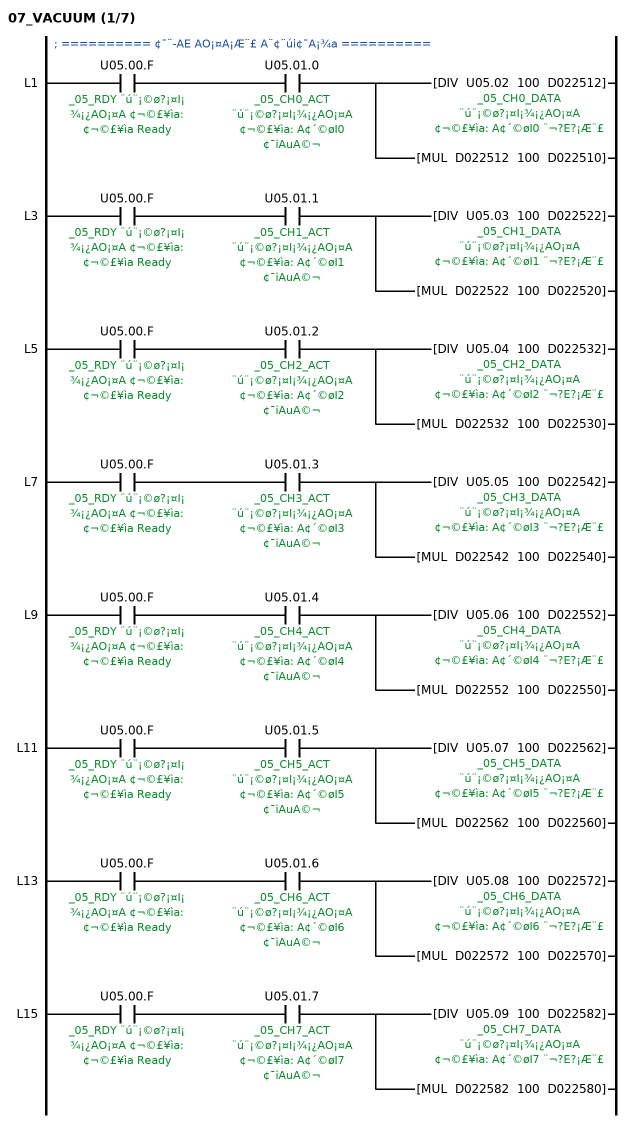
[picture p48: 07_VACUUM rungs L1-L15]
// ========== ¢¯¨­AE AO¡¤A¡Æ¨£ A¨¢¨úi¢¯A¡¾a ==========
; L1
LOAD      U05.00.F	// _05_RDY ¨ú¨¡©ø?¡¤I¡¾¡¿AO¡¤A ¢¬©£¥ìa: ¢¬©£¥ìa Ready
AND       U05.01.0	// _05_CH0_ACT ¨ú¨¡©ø?¡¤I¡¾¡¿AO¡¤A ¢¬©£¥ìa: A¢´©øI0 ¢¯iAuA©¬
DIV       U05.02 100 D022512	// _05_CH0_DATA ¨ú¨¡©ø?¡¤I¡¾¡¿AO¡¤A ¢¬©£¥ìa: A¢´©øI0 ¨¬?E?¡Æ¨£
MUL       D022512 100 D022510
; L3
LOAD      U05.00.F	// _05_RDY ¨ú¨¡©ø?¡¤I¡¾¡¿AO¡¤A ¢¬©£¥ìa: ¢¬©£¥ìa Ready
AND       U05.01.1	// _05_CH1_ACT ¨ú¨¡©ø?¡¤I¡¾¡¿AO¡¤A ¢¬©£¥ìa: A¢´©øI1 ¢¯iAuA©¬
DIV       U05.03 100 D022522	// _05_CH1_DATA ¨ú¨¡©ø?¡¤I¡¾¡¿AO¡¤A ¢¬©£¥ìa: A¢´©øI1 ¨¬?E?¡Æ¨£
MUL       D022522 100 D022520
; L5
LOAD      U05.00.F	// _05_RDY ¨ú¨¡©ø?¡¤I¡¾¡¿AO¡¤A ¢¬©£¥ìa: ¢¬©£¥ìa Ready
AND       U05.01.2	// _05_CH2_ACT ¨ú¨¡©ø?¡¤I¡¾¡¿AO¡¤A ¢¬©£¥ìa: A¢´©øI2 ¢¯iAuA©¬
DIV       U05.04 100 D022532	// _05_CH2_DATA ¨ú¨¡©ø?¡¤I¡¾¡¿AO¡¤A ¢¬©£¥ìa: A¢´©øI2 ¨¬?E?¡Æ¨£
MUL       D022532 100 D022530
; L7
LOAD      U05.00.F	// _05_RDY ¨ú¨¡©ø?¡¤I¡¾¡¿AO¡¤A ¢¬©£¥ìa: ¢¬©£¥ìa Ready
AND       U05.01.3	// _05_CH3_ACT ¨ú¨¡©ø?¡¤I¡¾¡¿AO¡¤A ¢¬©£¥ìa: A¢´©øI3 ¢¯iAuA©¬
DIV       U05.05 100 D022542	// _05_CH3_DATA ¨ú¨¡©ø?¡¤I¡¾¡¿AO¡¤A ¢¬©£¥ìa: A¢´©øI3 ¨¬?E?¡Æ¨£
MUL       D022542 100 D022540
; L9
LOAD      U05.00.F	// _05_RDY ¨ú¨¡©ø?¡¤I¡¾¡¿AO¡¤A ¢¬©£¥ìa: ¢¬©£¥ìa Ready
AND       U05.01.4	// _05_CH4_ACT ¨ú¨¡©ø?¡¤I¡¾¡¿AO¡¤A ¢¬©£¥ìa: A¢´©øI4 ¢¯iAuA©¬
DIV       U05.06 100 D022552	// _05_CH4_DATA ¨ú¨¡©ø?¡¤I¡¾¡¿AO¡¤A ¢¬©£¥ìa: A¢´©øI4 ¨¬?E?¡Æ¨£
MUL       D022552 100 D022550
; L11
LOAD      U05.00.F	// _05_RDY ¨ú¨¡©ø?¡¤I¡¾¡¿AO¡¤A ¢¬©£¥ìa: ¢¬©£¥ìa Ready
AND       U05.01.5	// _05_CH5_ACT ¨ú¨¡©ø?¡¤I¡¾¡¿AO¡¤A ¢¬©£¥ìa: A¢´©øI5 ¢¯iAuA©¬
DIV       U05.07 100 D022562	// _05_CH5_DATA ¨ú¨¡©ø?¡¤I¡¾¡¿AO¡¤A ¢¬©£¥ìa: A¢´©øI5 ¨¬?E?¡Æ¨£
MUL       D022562 100 D022560
; L13
LOAD      U05.00.F	// _05_RDY ¨ú¨¡©ø?¡¤I¡¾¡¿AO¡¤A ¢¬©£¥ìa: ¢¬©£¥ìa Ready
AND       U05.01.6	// _05_CH6_ACT ¨ú¨¡©ø?¡¤I¡¾¡¿AO¡¤A ¢¬©£¥ìa: A¢´©øI6 ¢¯iAuA©¬
DIV       U05.08 100 D022572	// _05_CH6_DATA ¨ú¨¡©ø?¡¤I¡¾¡¿AO¡¤A ¢¬©£¥ìa: A¢´©øI6 ¨¬?E?¡Æ¨£
MUL       D022572 100 D022570
; L15
LOAD      U05.00.F	// _05_RDY ¨ú¨¡©ø?¡¤I¡¾¡¿AO¡¤A ¢¬©£¥ìa: ¢¬©£¥ìa Ready
AND       U05.01.7	// _05_CH7_ACT ¨ú¨¡©ø?¡¤I¡¾¡¿AO¡¤A ¢¬©£¥ìa: A¢´©øI7 ¢¯iAuA©¬
DIV       U05.09 100 D022582	// _05_CH7_DATA ¨ú¨¡©ø?¡¤I¡¾¡¿AO¡¤A ¢¬©£¥ìa: A¢´©øI7 ¨¬?E?¡Æ¨£
MUL       D022582 100 D022580

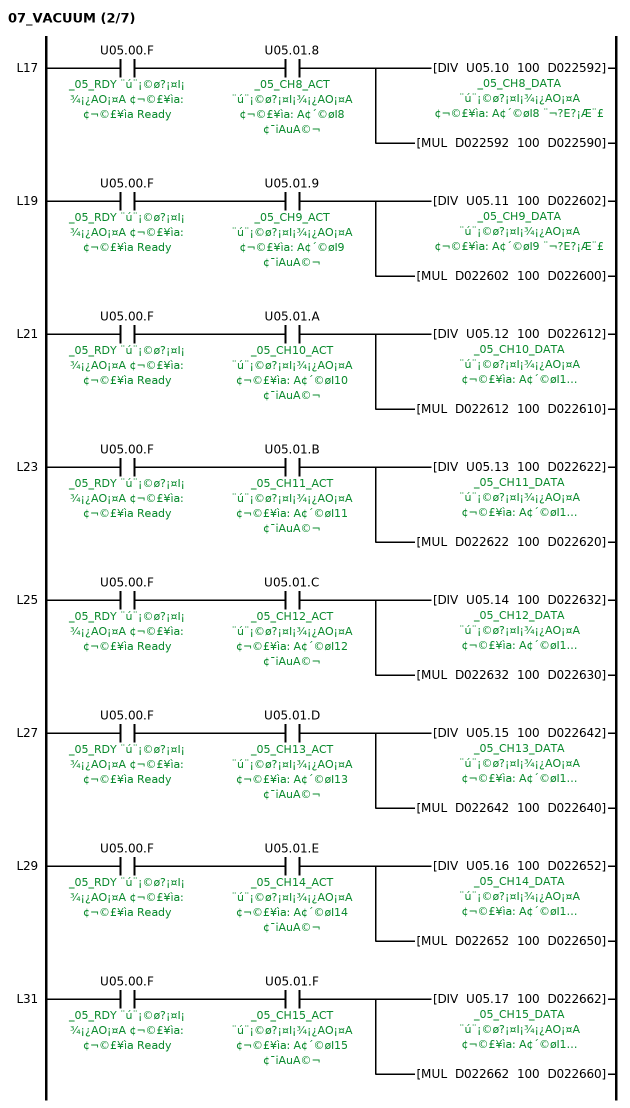
; L17
LOAD      U05.00.F	// _05_RDY ¨ú¨¡©ø?¡¤I¡¾¡¿AO¡¤A ¢¬©£¥ìa: ¢¬©£¥ìa Ready
AND       U05.01.8	// _05_CH8_ACT ¨ú¨¡©ø?¡¤I¡¾¡¿AO¡¤A ¢¬©£¥ìa: A¢´©øI8 ¢¯iAuA©¬
DIV       U05.10 100 D022592	// _05_CH8_DATA ¨ú¨¡©ø?¡¤I¡¾¡¿AO¡¤A ¢¬©£¥ìa: A¢´©øI8 ¨¬?E?¡Æ¨£
MUL       D022592 100 D022590
; L19
LOAD      U05.00.F	// _05_RDY ¨ú¨¡©ø?¡¤I¡¾¡¿AO¡¤A ¢¬©£¥ìa: ¢¬©£¥ìa Ready
AND       U05.01.9	// _05_CH9_ACT ¨ú¨¡©ø?¡¤I¡¾¡¿AO¡¤A ¢¬©£¥ìa: A¢´©øI9 ¢¯iAuA©¬
DIV       U05.11 100 D022602	// _05_CH9_DATA ¨ú¨¡©ø?¡¤I¡¾¡¿AO¡¤A ¢¬©£¥ìa: A¢´©øI9 ¨¬?E?¡Æ¨£
MUL       D022602 100 D022600
; L21
LOAD      U05.00.F	// _05_RDY ¨ú¨¡©ø?¡¤I¡¾¡¿AO¡¤A ¢¬©£¥ìa: ¢¬©£¥ìa Ready
AND       U05.01.A	// _05_CH10_ACT ¨ú¨¡©ø?¡¤I¡¾¡¿AO¡¤A ¢¬©£¥ìa: A¢´©øI10 ¢¯iAuA©¬
DIV       U05.12 100 D022612	// _05_CH10_DATA ¨ú¨¡©ø?¡¤I¡¾¡¿AO¡¤A ¢¬©£¥ìa: A¢´©øI10 ¨¬?E?¡Æ¨£
MUL       D022612 100 D022610
; L23
LOAD      U05.00.F	// _05_RDY ¨ú¨¡©ø?¡¤I¡¾¡¿AO¡¤A ¢¬©£¥ìa: ¢¬©£¥ìa Ready
AND       U05.01.B	// _05_CH11_ACT ¨ú¨¡©ø?¡¤I¡¾¡¿AO¡¤A ¢¬©£¥ìa: A¢´©øI11 ¢¯iAuA©¬
DIV       U05.13 100 D022622	// _05_CH11_DATA ¨ú¨¡©ø?¡¤I¡¾¡¿AO¡¤A ¢¬©£¥ìa: A¢´©øI11 ¨¬?E?¡Æ¨£
MUL       D022622 100 D022620
; L25
LOAD      U05.00.F	// _05_RDY ¨ú¨¡©ø?¡¤I¡¾¡¿AO¡¤A ¢¬©£¥ìa: ¢¬©£¥ìa Ready
AND       U05.01.C	// _05_CH12_ACT ¨ú¨¡©ø?¡¤I¡¾¡¿AO¡¤A ¢¬©£¥ìa: A¢´©øI12 ¢¯iAuA©¬
DIV       U05.14 100 D022632	// _05_CH12_DATA ¨ú¨¡©ø?¡¤I¡¾¡¿AO¡¤A ¢¬©£¥ìa: A¢´©øI12 ¨¬?E?¡Æ¨£
MUL       D022632 100 D022630
; L27
LOAD      U05.00.F	// _05_RDY ¨ú¨¡©ø?¡¤I¡¾¡¿AO¡¤A ¢¬©£¥ìa: ¢¬©£¥ìa Ready
AND       U05.01.D	// _05_CH13_ACT ¨ú¨¡©ø?¡¤I¡¾¡¿AO¡¤A ¢¬©£¥ìa: A¢´©øI13 ¢¯iAuA©¬
DIV       U05.15 100 D022642	// _05_CH13_DATA ¨ú¨¡©ø?¡¤I¡¾¡¿AO¡¤A ¢¬©£¥ìa: A¢´©øI13 ¨¬?E?¡Æ¨£
MUL       D022642 100 D022640
; L29
LOAD      U05.00.F	// _05_RDY ¨ú¨¡©ø?¡¤I¡¾¡¿AO¡¤A ¢¬©£¥ìa: ¢¬©£¥ìa Ready
AND       U05.01.E	// _05_CH14_ACT ¨ú¨¡©ø?¡¤I¡¾¡¿AO¡¤A ¢¬©£¥ìa: A¢´©øI14 ¢¯iAuA©¬
DIV       U05.16 100 D022652	// _05_CH14_DATA ¨ú¨¡©ø?¡¤I¡¾¡¿AO¡¤A ¢¬©£¥ìa: A¢´©øI14 ¨¬?E?¡Æ¨£
MUL       D022652 100 D022650
; L31
LOAD      U05.00.F	// _05_RDY ¨ú¨¡©ø?¡¤I¡¾¡¿AO¡¤A ¢¬©£¥ìa: ¢¬©£¥ìa Ready
AND       U05.01.F	// _05_CH15_ACT ¨ú¨¡©ø?¡¤I¡¾¡¿AO¡¤A ¢¬©£¥ìa: A¢´©øI15 ¢¯iAuA©¬
DIV       U05.17 100 D022662	// _05_CH15_DATA ¨ú¨¡©ø?¡¤I¡¾¡¿AO¡¤A ¢¬©£¥ìa: A¢´©øI15 ¨¬?E?¡Æ¨£
MUL       D022662 100 D022660

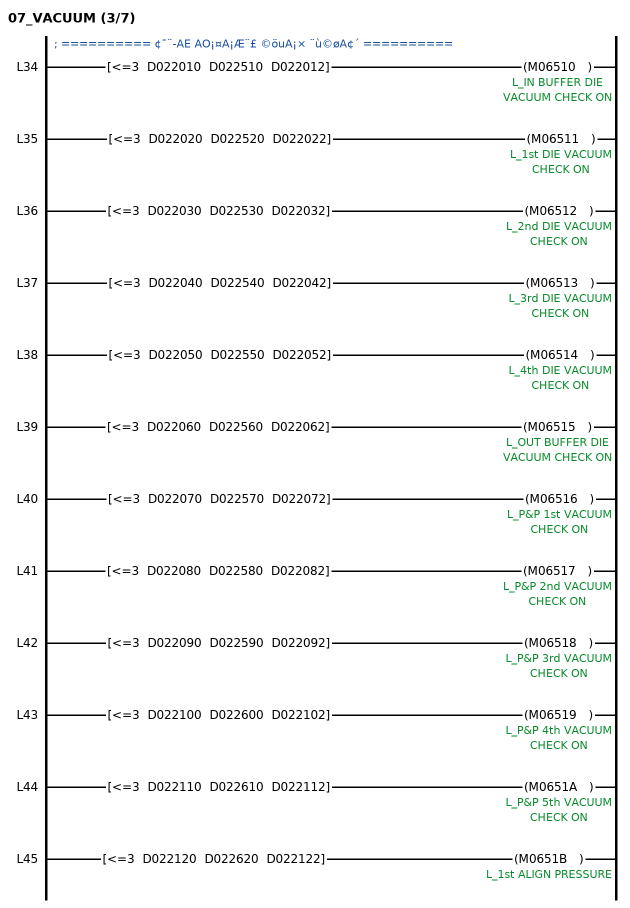
// ========== ¢¯¨­AE AO¡¤A¡Æ¨£ ©öuA¡× ¨ù©øA¢´ ==========
; L34
LOAD<=3   D022010 D022510 D022012
OUT       M06510	// L_IN BUFFER DIE VACUUM CHECK ON
; L35
LOAD<=3   D022020 D022520 D022022
OUT       M06511	// L_1st DIE VACUUM CHECK ON
; L36
LOAD<=3   D022030 D022530 D022032
OUT       M06512	// L_2nd DIE VACUUM CHECK ON
; L37
LOAD<=3   D022040 D022540 D022042
OUT       M06513	// L_3rd DIE VACUUM CHECK ON
; L38
LOAD<=3   D022050 D022550 D022052
OUT       M06514	// L_4th DIE VACUUM CHECK ON
; L39
LOAD<=3   D022060 D022560 D022062
OUT       M06515	// L_OUT BUFFER DIE VACUUM CHECK ON
; L40
LOAD<=3   D022070 D022570 D022072
OUT       M06516	// L_P&P 1st VACUUM CHECK ON
; L41
LOAD<=3   D022080 D022580 D022082
OUT       M06517	// L_P&P 2nd VACUUM CHECK ON
; L42
LOAD<=3   D022090 D022590 D022092
OUT       M06518	// L_P&P 3rd VACUUM CHECK ON
; L43
LOAD<=3   D022100 D022600 D022102
OUT       M06519	// L_P&P 4th VACUUM CHECK ON
; L44
LOAD<=3   D022110 D022610 D022112
OUT       M0651A	// L_P&P 5th VACUUM CHECK ON
; L45
LOAD<=3   D022120 D022620 D022122
OUT       M0651B	// L_1st ALIGN PRESSURE

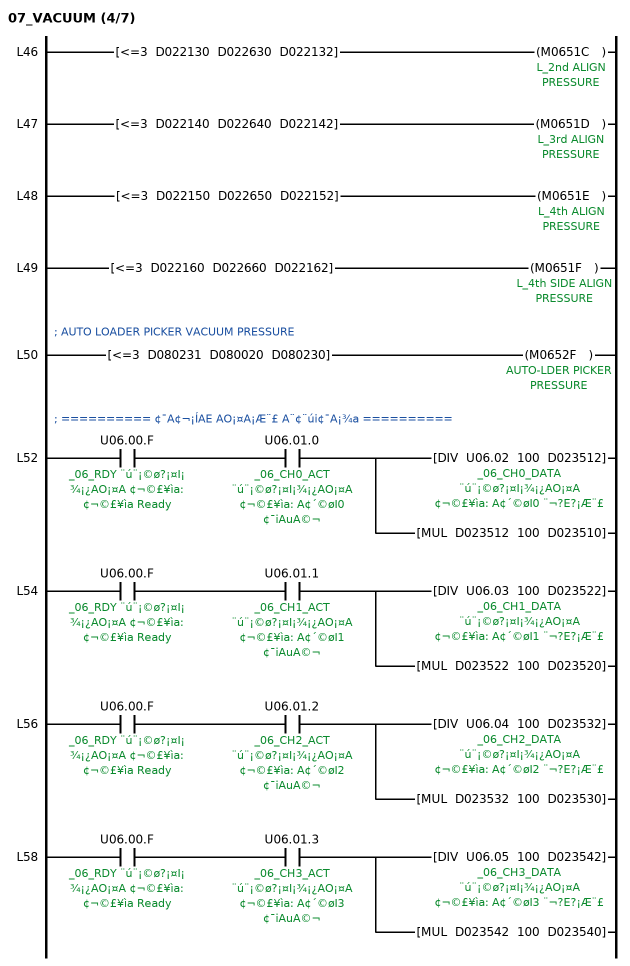
; L46
LOAD<=3   D022130 D022630 D022132
OUT       M0651C	// L_2nd ALIGN PRESSURE
; L47
LOAD<=3   D022140 D022640 D022142
OUT       M0651D	// L_3rd ALIGN PRESSURE
; L48
LOAD<=3   D022150 D022650 D022152
OUT       M0651E	// L_4th ALIGN PRESSURE
; L49
LOAD<=3   D022160 D022660 D022162
OUT       M0651F	// L_4th SIDE ALIGN PRESSURE
; L50
LOAD<=3   D080231 D080020 D080230
OUT       M0652F	// AUTO-LDER PICKER PRESSURE
// output comment: AUTO LOADER PICKER VACUUM PRESSURE
// ========== ¢¯A¢¬¡ÍAE AO¡¤A¡Æ¨£ A¨¢¨úi¢¯A¡¾a ==========
; L52
LOAD      U06.00.F	// _06_RDY ¨ú¨¡©ø?¡¤I¡¾¡¿AO¡¤A ¢¬©£¥ìa: ¢¬©£¥ìa Ready
AND       U06.01.0	// _06_CH0_ACT ¨ú¨¡©ø?¡¤I¡¾¡¿AO¡¤A ¢¬©£¥ìa: A¢´©øI0 ¢¯iAuA©¬
DIV       U06.02 100 D023512	// _06_CH0_DATA ¨ú¨¡©ø?¡¤I¡¾¡¿AO¡¤A ¢¬©£¥ìa: A¢´©øI0 ¨¬?E?¡Æ¨£
MUL       D023512 100 D023510
; L54
LOAD      U06.00.F	// _06_RDY ¨ú¨¡©ø?¡¤I¡¾¡¿AO¡¤A ¢¬©£¥ìa: ¢¬©£¥ìa Ready
AND       U06.01.1	// _06_CH1_ACT ¨ú¨¡©ø?¡¤I¡¾¡¿AO¡¤A ¢¬©£¥ìa: A¢´©øI1 ¢¯iAuA©¬
DIV       U06.03 100 D023522	// _06_CH1_DATA ¨ú¨¡©ø?¡¤I¡¾¡¿AO¡¤A ¢¬©£¥ìa: A¢´©øI1 ¨¬?E?¡Æ¨£
MUL       D023522 100 D023520
; L56
LOAD      U06.00.F	// _06_RDY ¨ú¨¡©ø?¡¤I¡¾¡¿AO¡¤A ¢¬©£¥ìa: ¢¬©£¥ìa Ready
AND       U06.01.2	// _06_CH2_ACT ¨ú¨¡©ø?¡¤I¡¾¡¿AO¡¤A ¢¬©£¥ìa: A¢´©øI2 ¢¯iAuA©¬
DIV       U06.04 100 D023532	// _06_CH2_DATA ¨ú¨¡©ø?¡¤I¡¾¡¿AO¡¤A ¢¬©£¥ìa: A¢´©øI2 ¨¬?E?¡Æ¨£
MUL       D023532 100 D023530
; L58
LOAD      U06.00.F	// _06_RDY ¨ú¨¡©ø?¡¤I¡¾¡¿AO¡¤A ¢¬©£¥ìa: ¢¬©£¥ìa Ready
AND       U06.01.3	// _06_CH3_ACT ¨ú¨¡©ø?¡¤I¡¾¡¿AO¡¤A ¢¬©£¥ìa: A¢´©øI3 ¢¯iAuA©¬
DIV       U06.05 100 D023542	// _06_CH3_DATA ¨ú¨¡©ø?¡¤I¡¾¡¿AO¡¤A ¢¬©£¥ìa: A¢´©øI3 ¨¬?E?¡Æ¨£
MUL       D023542 100 D023540

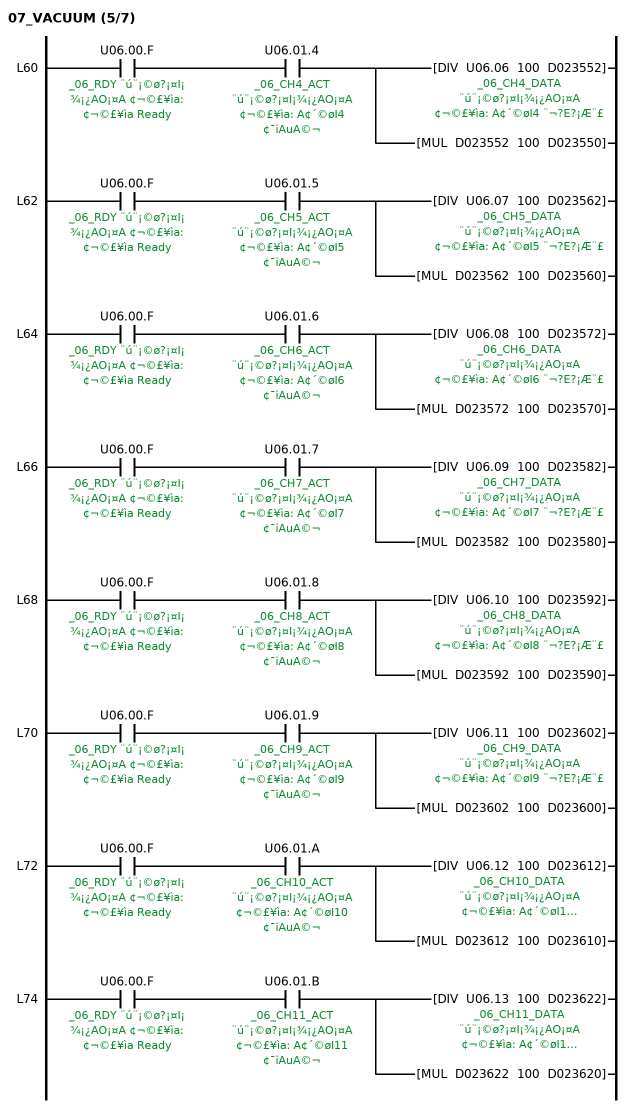
; L60
LOAD      U06.00.F	// _06_RDY ¨ú¨¡©ø?¡¤I¡¾¡¿AO¡¤A ¢¬©£¥ìa: ¢¬©£¥ìa Ready
AND       U06.01.4	// _06_CH4_ACT ¨ú¨¡©ø?¡¤I¡¾¡¿AO¡¤A ¢¬©£¥ìa: A¢´©øI4 ¢¯iAuA©¬
DIV       U06.06 100 D023552	// _06_CH4_DATA ¨ú¨¡©ø?¡¤I¡¾¡¿AO¡¤A ¢¬©£¥ìa: A¢´©øI4 ¨¬?E?¡Æ¨£
MUL       D023552 100 D023550
; L62
LOAD      U06.00.F	// _06_RDY ¨ú¨¡©ø?¡¤I¡¾¡¿AO¡¤A ¢¬©£¥ìa: ¢¬©£¥ìa Ready
AND       U06.01.5	// _06_CH5_ACT ¨ú¨¡©ø?¡¤I¡¾¡¿AO¡¤A ¢¬©£¥ìa: A¢´©øI5 ¢¯iAuA©¬
DIV       U06.07 100 D023562	// _06_CH5_DATA ¨ú¨¡©ø?¡¤I¡¾¡¿AO¡¤A ¢¬©£¥ìa: A¢´©øI5 ¨¬?E?¡Æ¨£
MUL       D023562 100 D023560
; L64
LOAD      U06.00.F	// _06_RDY ¨ú¨¡©ø?¡¤I¡¾¡¿AO¡¤A ¢¬©£¥ìa: ¢¬©£¥ìa Ready
AND       U06.01.6	// _06_CH6_ACT ¨ú¨¡©ø?¡¤I¡¾¡¿AO¡¤A ¢¬©£¥ìa: A¢´©øI6 ¢¯iAuA©¬
DIV       U06.08 100 D023572	// _06_CH6_DATA ¨ú¨¡©ø?¡¤I¡¾¡¿AO¡¤A ¢¬©£¥ìa: A¢´©øI6 ¨¬?E?¡Æ¨£
MUL       D023572 100 D023570
; L66
LOAD      U06.00.F	// _06_RDY ¨ú¨¡©ø?¡¤I¡¾¡¿AO¡¤A ¢¬©£¥ìa: ¢¬©£¥ìa Ready
AND       U06.01.7	// _06_CH7_ACT ¨ú¨¡©ø?¡¤I¡¾¡¿AO¡¤A ¢¬©£¥ìa: A¢´©øI7 ¢¯iAuA©¬
DIV       U06.09 100 D023582	// _06_CH7_DATA ¨ú¨¡©ø?¡¤I¡¾¡¿AO¡¤A ¢¬©£¥ìa: A¢´©øI7 ¨¬?E?¡Æ¨£
MUL       D023582 100 D023580
; L68
LOAD      U06.00.F	// _06_RDY ¨ú¨¡©ø?¡¤I¡¾¡¿AO¡¤A ¢¬©£¥ìa: ¢¬©£¥ìa Ready
AND       U06.01.8	// _06_CH8_ACT ¨ú¨¡©ø?¡¤I¡¾¡¿AO¡¤A ¢¬©£¥ìa: A¢´©øI8 ¢¯iAuA©¬
DIV       U06.10 100 D023592	// _06_CH8_DATA ¨ú¨¡©ø?¡¤I¡¾¡¿AO¡¤A ¢¬©£¥ìa: A¢´©øI8 ¨¬?E?¡Æ¨£
MUL       D023592 100 D023590
; L70
LOAD      U06.00.F	// _06_RDY ¨ú¨¡©ø?¡¤I¡¾¡¿AO¡¤A ¢¬©£¥ìa: ¢¬©£¥ìa Ready
AND       U06.01.9	// _06_CH9_ACT ¨ú¨¡©ø?¡¤I¡¾¡¿AO¡¤A ¢¬©£¥ìa: A¢´©øI9 ¢¯iAuA©¬
DIV       U06.11 100 D023602	// _06_CH9_DATA ¨ú¨¡©ø?¡¤I¡¾¡¿AO¡¤A ¢¬©£¥ìa: A¢´©øI9 ¨¬?E?¡Æ¨£
MUL       D023602 100 D023600
; L72
LOAD      U06.00.F	// _06_RDY ¨ú¨¡©ø?¡¤I¡¾¡¿AO¡¤A ¢¬©£¥ìa: ¢¬©£¥ìa Ready
AND       U06.01.A	// _06_CH10_ACT ¨ú¨¡©ø?¡¤I¡¾¡¿AO¡¤A ¢¬©£¥ìa: A¢´©øI10 ¢¯iAuA©¬
DIV       U06.12 100 D023612	// _06_CH10_DATA ¨ú¨¡©ø?¡¤I¡¾¡¿AO¡¤A ¢¬©£¥ìa: A¢´©øI10 ¨¬?E?¡Æ¨£
MUL       D023612 100 D023610
; L74
LOAD      U06.00.F	// _06_RDY ¨ú¨¡©ø?¡¤I¡¾¡¿AO¡¤A ¢¬©£¥ìa: ¢¬©£¥ìa Ready
AND       U06.01.B	// _06_CH11_ACT ¨ú¨¡©ø?¡¤I¡¾¡¿AO¡¤A ¢¬©£¥ìa: A¢´©øI11 ¢¯iAuA©¬
DIV       U06.13 100 D023622	// _06_CH11_DATA ¨ú¨¡©ø?¡¤I¡¾¡¿AO¡¤A ¢¬©£¥ìa: A¢´©øI11 ¨¬?E?¡Æ¨£
MUL       D023622 100 D023620

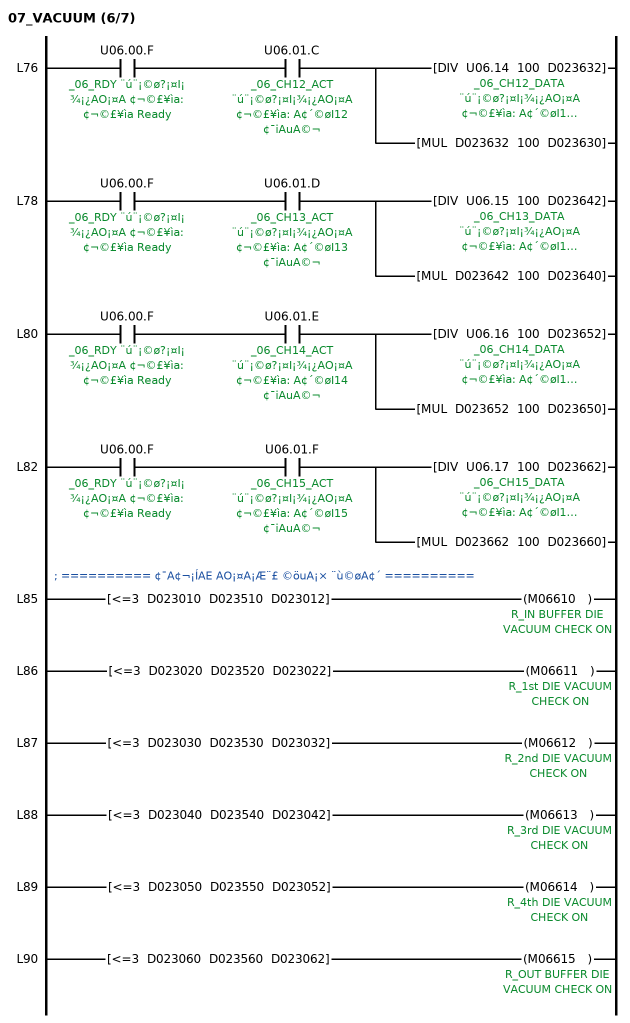
; L76
LOAD      U06.00.F	// _06_RDY ¨ú¨¡©ø?¡¤I¡¾¡¿AO¡¤A ¢¬©£¥ìa: ¢¬©£¥ìa Ready
AND       U06.01.C	// _06_CH12_ACT ¨ú¨¡©ø?¡¤I¡¾¡¿AO¡¤A ¢¬©£¥ìa: A¢´©øI12 ¢¯iAuA©¬
DIV       U06.14 100 D023632	// _06_CH12_DATA ¨ú¨¡©ø?¡¤I¡¾¡¿AO¡¤A ¢¬©£¥ìa: A¢´©øI12 ¨¬?E?¡Æ¨£
MUL       D023632 100 D023630
; L78
LOAD      U06.00.F	// _06_RDY ¨ú¨¡©ø?¡¤I¡¾¡¿AO¡¤A ¢¬©£¥ìa: ¢¬©£¥ìa Ready
AND       U06.01.D	// _06_CH13_ACT ¨ú¨¡©ø?¡¤I¡¾¡¿AO¡¤A ¢¬©£¥ìa: A¢´©øI13 ¢¯iAuA©¬
DIV       U06.15 100 D023642	// _06_CH13_DATA ¨ú¨¡©ø?¡¤I¡¾¡¿AO¡¤A ¢¬©£¥ìa: A¢´©øI13 ¨¬?E?¡Æ¨£
MUL       D023642 100 D023640
; L80
LOAD      U06.00.F	// _06_RDY ¨ú¨¡©ø?¡¤I¡¾¡¿AO¡¤A ¢¬©£¥ìa: ¢¬©£¥ìa Ready
AND       U06.01.E	// _06_CH14_ACT ¨ú¨¡©ø?¡¤I¡¾¡¿AO¡¤A ¢¬©£¥ìa: A¢´©øI14 ¢¯iAuA©¬
DIV       U06.16 100 D023652	// _06_CH14_DATA ¨ú¨¡©ø?¡¤I¡¾¡¿AO¡¤A ¢¬©£¥ìa: A¢´©øI14 ¨¬?E?¡Æ¨£
MUL       D023652 100 D023650
; L82
LOAD      U06.00.F	// _06_RDY ¨ú¨¡©ø?¡¤I¡¾¡¿AO¡¤A ¢¬©£¥ìa: ¢¬©£¥ìa Ready
AND       U06.01.F	// _06_CH15_ACT ¨ú¨¡©ø?¡¤I¡¾¡¿AO¡¤A ¢¬©£¥ìa: A¢´©øI15 ¢¯iAuA©¬
DIV       U06.17 100 D023662	// _06_CH15_DATA ¨ú¨¡©ø?¡¤I¡¾¡¿AO¡¤A ¢¬©£¥ìa: A¢´©øI15 ¨¬?E?¡Æ¨£
MUL       D023662 100 D023660
// ========== ¢¯A¢¬¡ÍAE AO¡¤A¡Æ¨£ ©öuA¡× ¨ù©øA¢´ ==========
; L85
LOAD<=3   D023010 D023510 D023012
OUT       M06610	// R_IN BUFFER DIE VACUUM CHECK ON
; L86
LOAD<=3   D023020 D023520 D023022
OUT       M06611	// R_1st DIE VACUUM CHECK ON
; L87
LOAD<=3   D023030 D023530 D023032
OUT       M06612	// R_2nd DIE VACUUM CHECK ON
; L88
LOAD<=3   D023040 D023540 D023042
OUT       M06613	// R_3rd DIE VACUUM CHECK ON
; L89
LOAD<=3   D023050 D023550 D023052
OUT       M06614	// R_4th DIE VACUUM CHECK ON
; L90
LOAD<=3   D023060 D023560 D023062
OUT       M06615	// R_OUT BUFFER DIE VACUUM CHECK ON

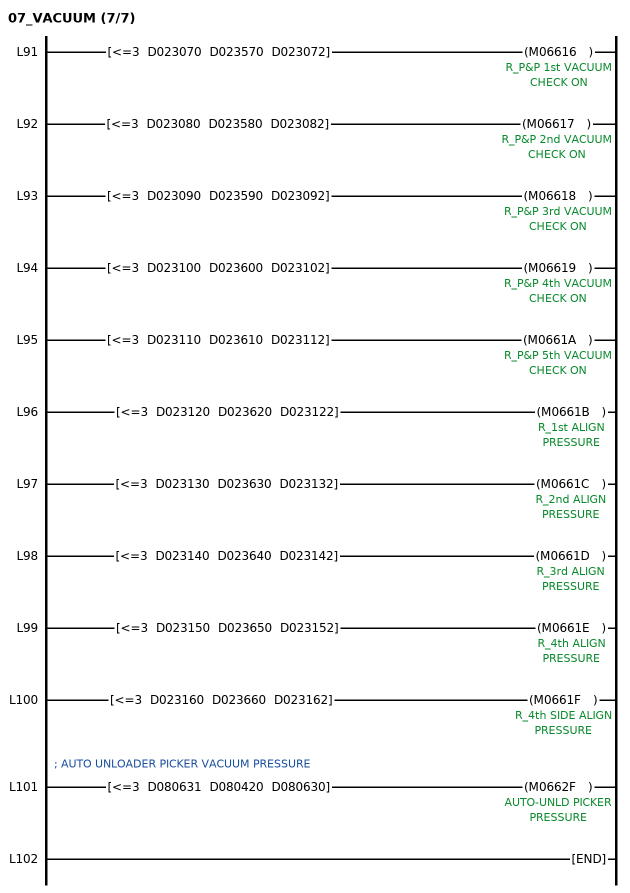
; L91
LOAD<=3   D023070 D023570 D023072
OUT       M06616	// R_P&P 1st VACUUM CHECK ON
; L92
LOAD<=3   D023080 D023580 D023082
OUT       M06617	// R_P&P 2nd VACUUM CHECK ON
; L93
LOAD<=3   D023090 D023590 D023092
OUT       M06618	// R_P&P 3rd VACUUM CHECK ON
; L94
LOAD<=3   D023100 D023600 D023102
OUT       M06619	// R_P&P 4th VACUUM CHECK ON
; L95
LOAD<=3   D023110 D023610 D023112
OUT       M0661A	// R_P&P 5th VACUUM CHECK ON
; L96
LOAD<=3   D023120 D023620 D023122
OUT       M0661B	// R_1st ALIGN PRESSURE
; L97
LOAD<=3   D023130 D023630 D023132
OUT       M0661C	// R_2nd ALIGN PRESSURE
; L98
LOAD<=3   D023140 D023640 D023142
OUT       M0661D	// R_3rd ALIGN PRESSURE
; L99
LOAD<=3   D023150 D023650 D023152
OUT       M0661E	// R_4th ALIGN PRESSURE
; L100
LOAD<=3   D023160 D023660 D023162
OUT       M0661F	// R_4th SIDE ALIGN PRESSURE
; L101
LOAD<=3   D080631 D080420 D080630
OUT       M0662F	// AUTO-UNLD PICKER PRESSURE
// output comment: AUTO UNLOADER PICKER VACUUM PRESSURE
; L102
END

PROGRAM 11_L_1st_MAND (task: ¨ö¨¬A¥ì CA¡¤I¡¾¡¿¡¤¡Í)

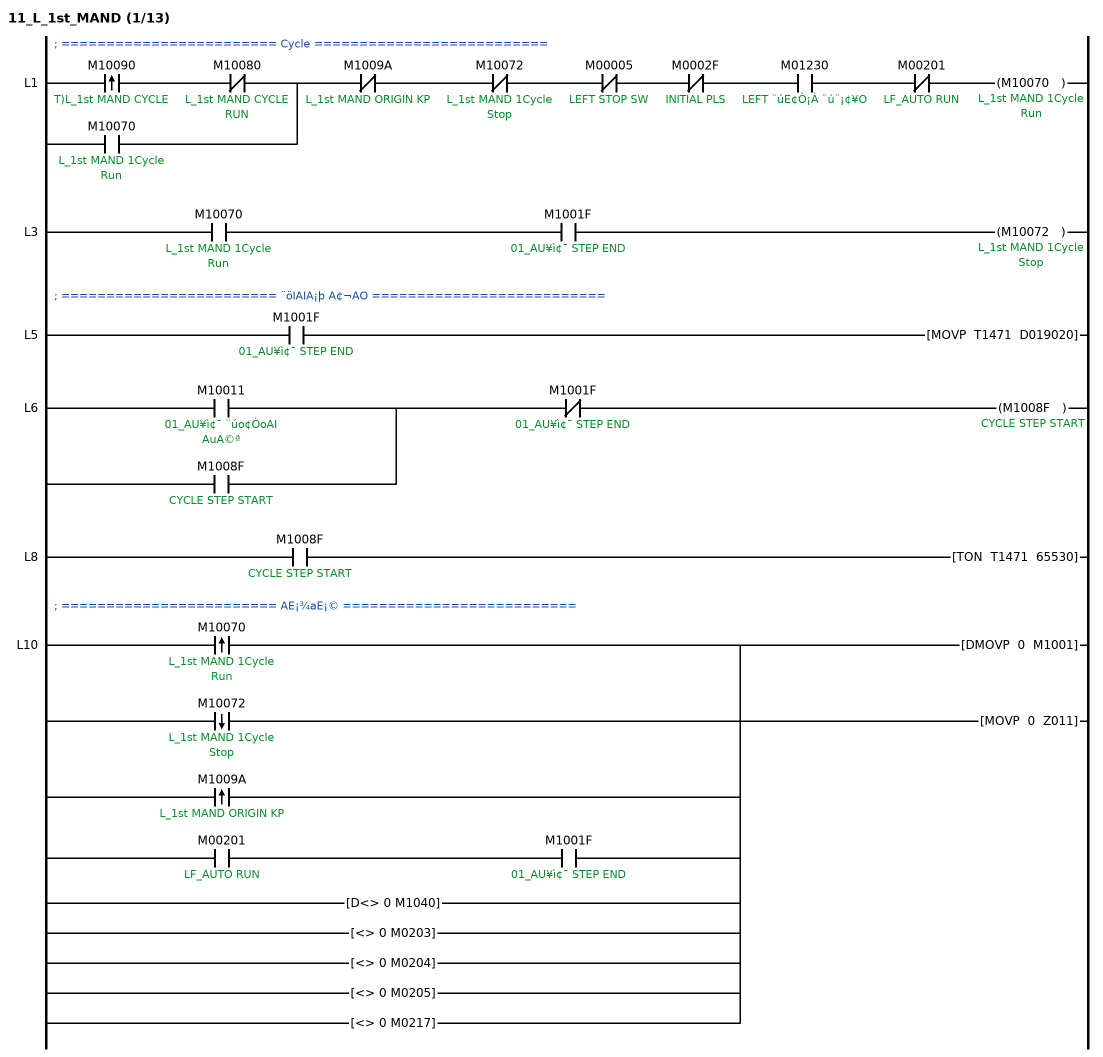
// ======================== Cycle ==========================
; L1
LOADP     M10090	// T)L_1st MAND CYCLE
AND NOT   M10080	// L_1st MAND CYCLE RUN
OR        M10070	// L_1st MAND 1Cycle Run
AND NOT   M1009A	// L_1st MAND ORIGIN KP
AND NOT   M10072	// L_1st MAND 1Cycle Stop
AND NOT   M00005	// LEFT STOP SW
AND NOT   M0002F	// INITIAL PLS
AND       M01230	// LEFT ¨úE¢Ò¡À ¨ú¨¡¢¥O
AND NOT   M00201	// LF_AUTO RUN
OUT       M10070	// L_1st MAND 1Cycle Run
; L3
LOAD      M10070	// L_1st MAND 1Cycle Run
AND       M1001F	// 01_AU¥ì¢¯ STEP END
OUT       M10072	// L_1st MAND 1Cycle Stop
// ======================== ¨öIAIA¡þ A¢¬AO ==========================
; L5
LOAD      M1001F	// 01_AU¥ì¢¯ STEP END
MOVP      T1471 D019020
; L6
LOAD      M10011	// 01_AU¥ì¢¯ ¨úo¢ÒoAI AuA©ª
OR        M1008F	// CYCLE STEP START
AND NOT   M1001F	// 01_AU¥ì¢¯ STEP END
OUT       M1008F	// CYCLE STEP START
; L8
LOAD      M1008F	// CYCLE STEP START
TON       T1471 65530
// ======================== AE¡¾aE¡© ==========================
; L10
LOADP     M10070	// L_1st MAND 1Cycle Run
ORN       M10072	// L_1st MAND 1Cycle Stop
ORP       M1009A	// L_1st MAND ORIGIN KP
LOAD      M00201	// LF_AUTO RUN
AND       M1001F	// 01_AU¥ì¢¯ STEP END
OR LOAD
ORD<>     0 M1040
OR<>      0 M0203
OR<>      0 M0204
OR<>      0 M0205
OR<>      0 M0217
DMOVP     0 M1001
MOVP      0 Z011

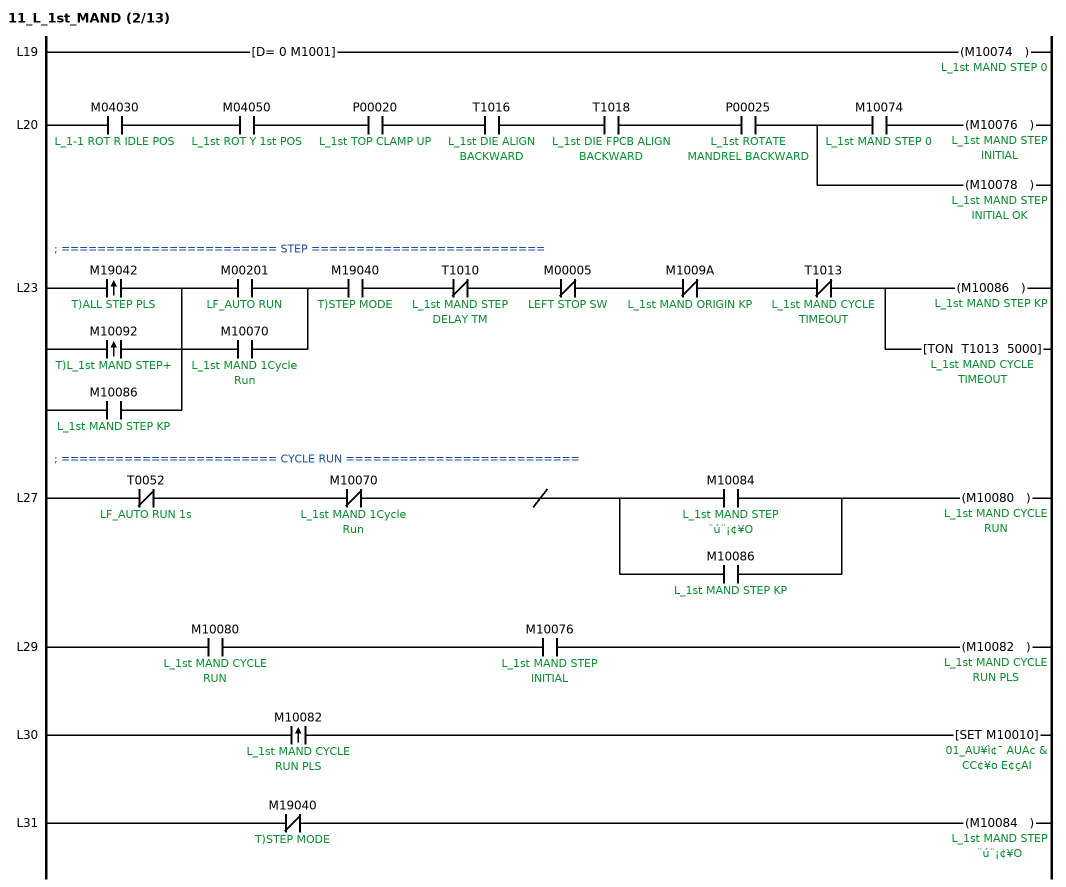
; L19
LOADD=    0 M1001
OUT       M10074	// L_1st MAND STEP 0
; L20
LOAD      M04030	// L_1-1 ROT R IDLE POS
AND       M04050	// L_1st ROT Y 1st POS
AND       P00020	// L_1st TOP CLAMP UP
AND       T1016	// L_1st DIE ALIGN BACKWARD
AND       T1018	// L_1st DIE FPCB ALIGN BACKWARD
AND       P00025	// L_1st ROTATE MANDREL BACKWARD
MPUSH
AND       M10074	// L_1st MAND STEP 0
OUT       M10076	// L_1st MAND STEP INITIAL
MPOP
OUT       M10078	// L_1st MAND STEP INITIAL OK
// ======================== STEP ==========================
; L23
LOADP     M19042	// T)ALL STEP PLS
ORP       M10092	// T)L_1st MAND STEP+
OR        M10086	// L_1st MAND STEP KP
LOAD      M00201	// LF_AUTO RUN
OR        M10070	// L_1st MAND 1Cycle Run
AND LOAD
AND       M19040	// T)STEP MODE
AND NOT   T1010	// L_1st MAND STEP DELAY TM
AND NOT   M00005	// LEFT STOP SW
AND NOT   M1009A	// L_1st MAND ORIGIN KP
AND NOT   T1013	// L_1st MAND CYCLE TIMEOUT
OUT       M10086	// L_1st MAND STEP KP
TON       T1013 5000	// L_1st MAND CYCLE TIMEOUT
// ======================== CYCLE RUN ==========================
; L27
LOAD NOT  T0052	// LF_AUTO RUN 1s
AND NOT   M10070	// L_1st MAND 1Cycle Run
NOT
LOAD      M10084	// L_1st MAND STEP ¨ú¨¡¢¥O
OR        M10086	// L_1st MAND STEP KP
AND LOAD
OUT       M10080	// L_1st MAND CYCLE RUN
; L29
LOAD      M10080	// L_1st MAND CYCLE RUN
AND       M10076	// L_1st MAND STEP INITIAL
OUT       M10082	// L_1st MAND CYCLE RUN PLS
; L30
LOADP     M10082	// L_1st MAND CYCLE RUN PLS
SET       M10010	// 01_AU¥ì¢¯ AUAc & CC¢¥o E¢çAI
; L31
LOAD NOT  M19040	// T)STEP MODE
OUT       M10084	// L_1st MAND STEP ¨ú¨¡¢¥O

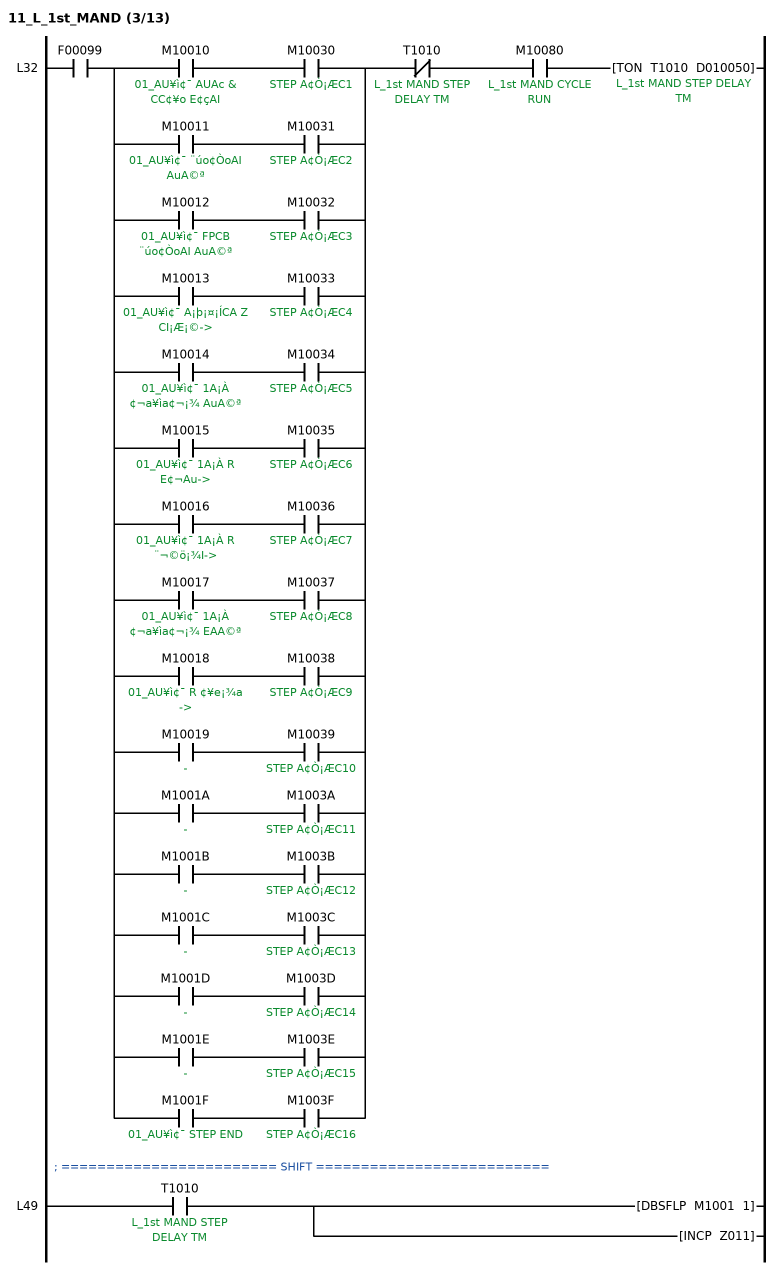
; L32
LOAD      F00099
LOAD      M10010	// 01_AU¥ì¢¯ AUAc & CC¢¥o E¢çAI
AND       M10030	// STEP A¢Ò¡ÆC1
LOAD      M10011	// 01_AU¥ì¢¯ ¨úo¢ÒoAI AuA©ª
AND       M10031	// STEP A¢Ò¡ÆC2
OR LOAD
LOAD      M10012	// 01_AU¥ì¢¯ FPCB ¨úo¢ÒoAI AuA©ª
AND       M10032	// STEP A¢Ò¡ÆC3
OR LOAD
LOAD      M10013	// 01_AU¥ì¢¯ A¡þ¡¤¡ÍCA Z CI¡Æ¡©->
AND       M10033	// STEP A¢Ò¡ÆC4
OR LOAD
LOAD      M10014	// 01_AU¥ì¢¯ 1A¡À ¢¬a¥ìa¢¬¡¾ AuA©ª
AND       M10034	// STEP A¢Ò¡ÆC5
OR LOAD
LOAD      M10015	// 01_AU¥ì¢¯ 1A¡À R E¢¬Au->
AND       M10035	// STEP A¢Ò¡ÆC6
OR LOAD
LOAD      M10016	// 01_AU¥ì¢¯ 1A¡À R ¨¬©ö¡¾I->
AND       M10036	// STEP A¢Ò¡ÆC7
OR LOAD
LOAD      M10017	// 01_AU¥ì¢¯ 1A¡À ¢¬a¥ìa¢¬¡¾ EAA©ª
AND       M10037	// STEP A¢Ò¡ÆC8
OR LOAD
LOAD      M10018	// 01_AU¥ì¢¯ R ¢¥e¡¾a ->
AND       M10038	// STEP A¢Ò¡ÆC9
OR LOAD
LOAD      M10019	// -
AND       M10039	// STEP A¢Ò¡ÆC10
OR LOAD
LOAD      M1001A	// -
AND       M1003A	// STEP A¢Ò¡ÆC11
OR LOAD
LOAD      M1001B	// -
AND       M1003B	// STEP A¢Ò¡ÆC12
OR LOAD
LOAD      M1001C	// -
AND       M1003C	// STEP A¢Ò¡ÆC13
OR LOAD
LOAD      M1001D	// -
AND       M1003D	// STEP A¢Ò¡ÆC14
OR LOAD
LOAD      M1001E	// -
AND       M1003E	// STEP A¢Ò¡ÆC15
OR LOAD
LOAD      M1001F	// 01_AU¥ì¢¯ STEP END
AND       M1003F	// STEP A¢Ò¡ÆC16
OR LOAD
AND LOAD
AND NOT   T1010	// L_1st MAND STEP DELAY TM
AND       M10080	// L_1st MAND CYCLE RUN
TON       T1010 D010050	// L_1st MAND STEP DELAY TM
// ======================== SHIFT ==========================
; L49
LOAD      T1010	// L_1st MAND STEP DELAY TM
DBSFLP    M1001 1
INCP      Z011

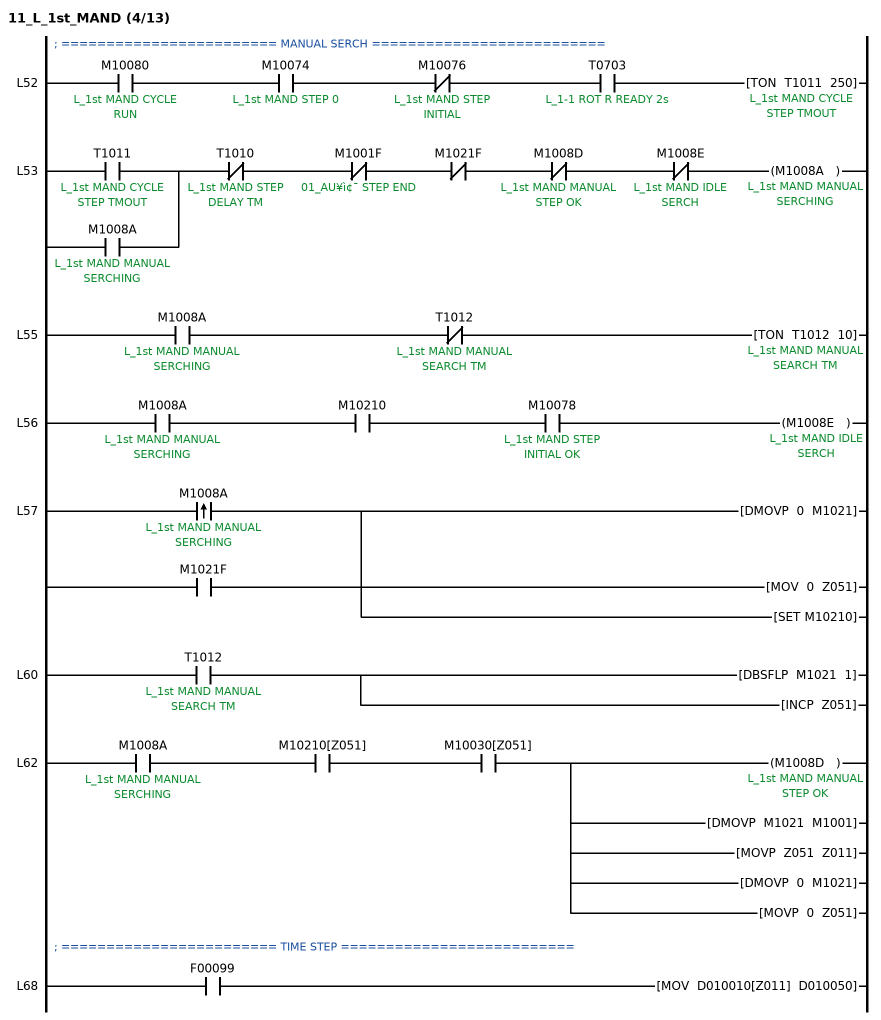
// ======================== MANUAL SERCH ==========================
; L52
LOAD      M10080	// L_1st MAND CYCLE RUN
AND       M10074	// L_1st MAND STEP 0
AND NOT   M10076	// L_1st MAND STEP INITIAL
AND       T0703	// L_1-1 ROT R READY 2s
TON       T1011 250	// L_1st MAND CYCLE STEP TMOUT
; L53
LOAD      T1011	// L_1st MAND CYCLE STEP TMOUT
OR        M1008A	// L_1st MAND MANUAL SERCHING
AND NOT   T1010	// L_1st MAND STEP DELAY TM
AND NOT   M1001F	// 01_AU¥ì¢¯ STEP END
AND NOT   M1021F
AND NOT   M1008D	// L_1st MAND MANUAL STEP OK
AND NOT   M1008E	// L_1st MAND IDLE SERCH
OUT       M1008A	// L_1st MAND MANUAL SERCHING
; L55
LOAD      M1008A	// L_1st MAND MANUAL SERCHING
AND NOT   T1012	// L_1st MAND MANUAL SEARCH TM
TON       T1012 10	// L_1st MAND MANUAL SEARCH TM
; L56
LOAD      M1008A	// L_1st MAND MANUAL SERCHING
AND       M10210
AND       M10078	// L_1st MAND STEP INITIAL OK
OUT       M1008E	// L_1st MAND IDLE SERCH
; L57
LOADP     M1008A	// L_1st MAND MANUAL SERCHING
OR        M1021F
DMOVP     0 M1021
MOV       0 Z051
SET       M10210
; L60
LOAD      T1012	// L_1st MAND MANUAL SEARCH TM
DBSFLP    M1021 1
INCP      Z051
; L62
LOAD      M1008A	// L_1st MAND MANUAL SERCHING
AND       M10210[Z051]
AND       M10030[Z051]
OUT       M1008D	// L_1st MAND MANUAL STEP OK
DMOVP     M1021 M1001
MOVP      Z051 Z011
DMOVP     0 M1021
MOVP      0 Z051
// ======================== TIME STEP ==========================
; L68
LOAD      F00099
MOV       D010010[Z011] D010050

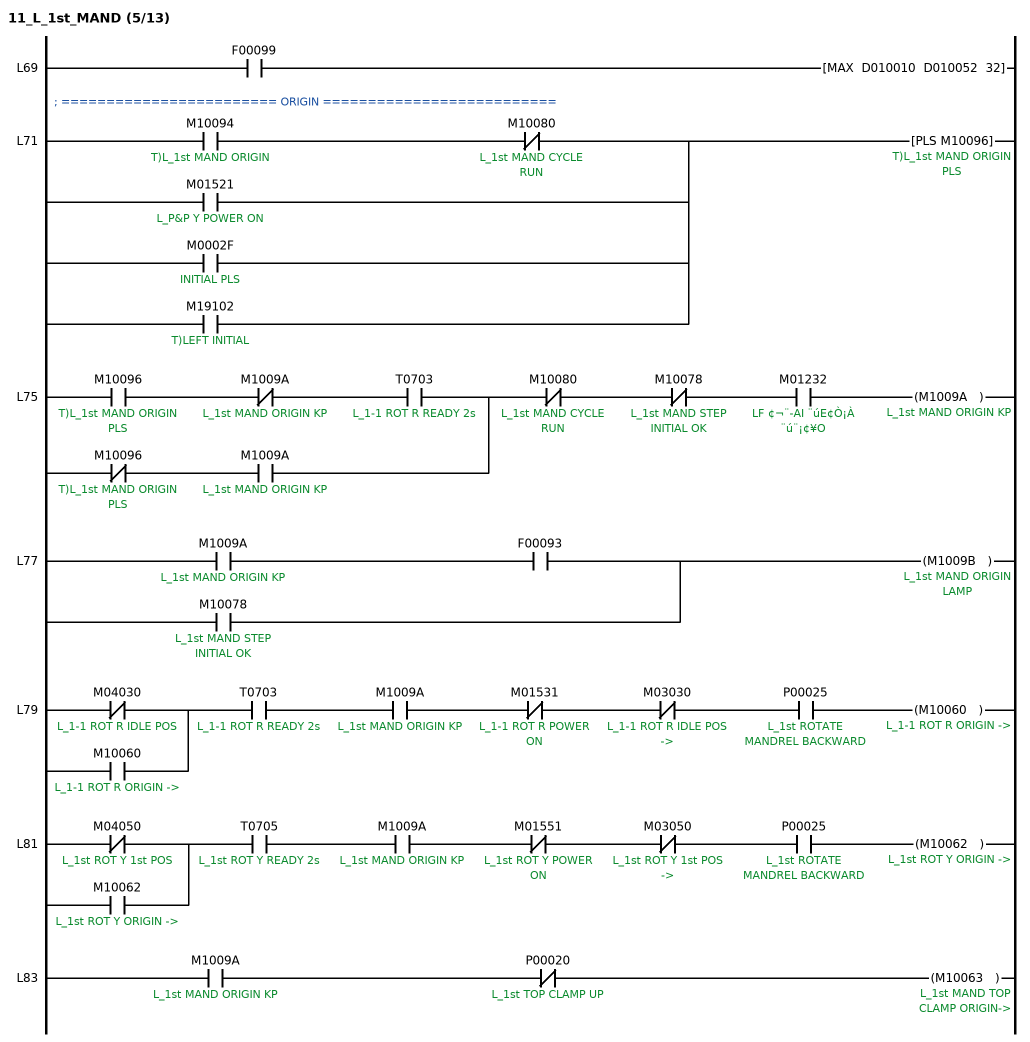
; L69
LOAD      F00099
MAX       D010010 D010052 32
// ======================== ORIGIN ==========================
; L71
LOAD      M10094	// T)L_1st MAND ORIGIN
AND NOT   M10080	// L_1st MAND CYCLE RUN
OR        M01521	// L_P&P Y POWER ON
OR        M0002F	// INITIAL PLS
OR        M19102	// T)LEFT INITIAL
OUTP      M10096	// T)L_1st MAND ORIGIN PLS
; L75
LOAD      M10096	// T)L_1st MAND ORIGIN PLS
AND NOT   M1009A	// L_1st MAND ORIGIN KP
AND       T0703	// L_1-1 ROT R READY 2s
LOAD NOT  M10096	// T)L_1st MAND ORIGIN PLS
AND       M1009A	// L_1st MAND ORIGIN KP
OR LOAD
AND NOT   M10080	// L_1st MAND CYCLE RUN
AND NOT   M10078	// L_1st MAND STEP INITIAL OK
AND       M01232	// LF ¢¬¨­AI ¨úE¢Ò¡À ¨ú¨¡¢¥O
OUT       M1009A	// L_1st MAND ORIGIN KP
; L77
LOAD      M1009A	// L_1st MAND ORIGIN KP
AND       F00093
OR        M10078	// L_1st MAND STEP INITIAL OK
OUT       M1009B	// L_1st MAND ORIGIN LAMP
; L79
LOAD NOT  M04030	// L_1-1 ROT R IDLE POS
OR        M10060	// L_1-1 ROT R ORIGIN ->
AND       T0703	// L_1-1 ROT R READY 2s
AND       M1009A	// L_1st MAND ORIGIN KP
AND NOT   M01531	// L_1-1 ROT R POWER ON
AND NOT   M03030	// L_1-1 ROT R IDLE POS ->
AND       P00025	// L_1st ROTATE MANDREL BACKWARD
OUT       M10060	// L_1-1 ROT R ORIGIN ->
; L81
LOAD NOT  M04050	// L_1st ROT Y 1st POS
OR        M10062	// L_1st ROT Y ORIGIN ->
AND       T0705	// L_1st ROT Y READY 2s
AND       M1009A	// L_1st MAND ORIGIN KP
AND NOT   M01551	// L_1st ROT Y POWER ON
AND NOT   M03050	// L_1st ROT Y 1st POS ->
AND       P00025	// L_1st ROTATE MANDREL BACKWARD
OUT       M10062	// L_1st ROT Y ORIGIN ->
; L83
LOAD      M1009A	// L_1st MAND ORIGIN KP
AND NOT   P00020	// L_1st TOP CLAMP UP
OUT       M10063	// L_1st MAND TOP CLAMP ORIGIN->

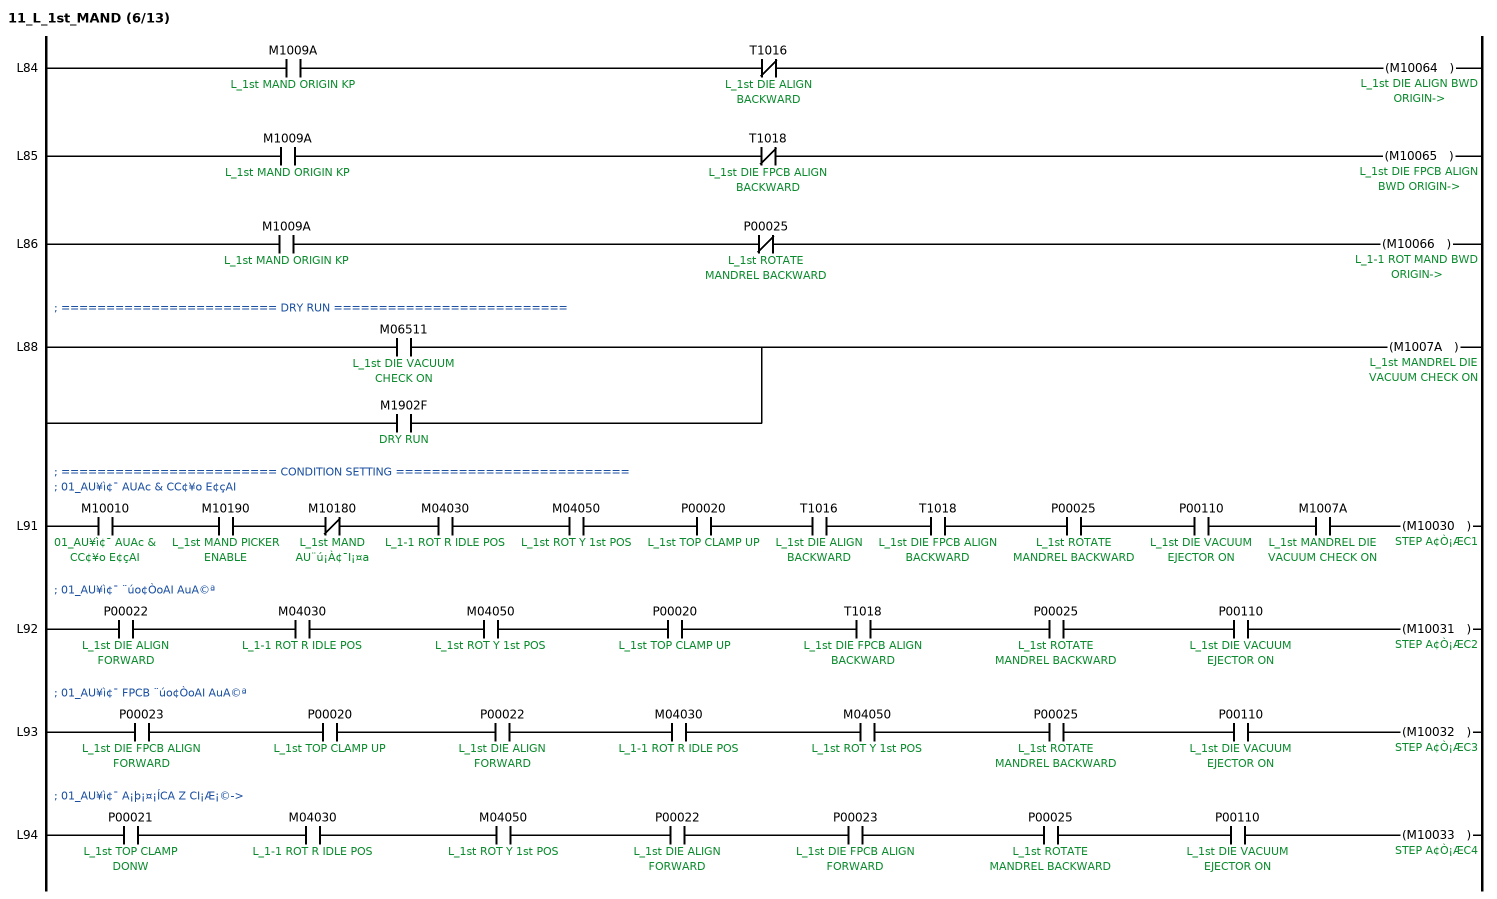
; L84
LOAD      M1009A	// L_1st MAND ORIGIN KP
AND NOT   T1016	// L_1st DIE ALIGN BACKWARD
OUT       M10064	// L_1st DIE ALIGN BWD ORIGIN->
; L85
LOAD      M1009A	// L_1st MAND ORIGIN KP
AND NOT   T1018	// L_1st DIE FPCB ALIGN BACKWARD
OUT       M10065	// L_1st DIE FPCB ALIGN BWD ORIGIN->
; L86
LOAD      M1009A	// L_1st MAND ORIGIN KP
AND NOT   P00025	// L_1st ROTATE MANDREL BACKWARD
OUT       M10066	// L_1-1 ROT MAND BWD ORIGIN->
// ======================== DRY RUN ==========================
; L88
LOAD      M06511	// L_1st DIE VACUUM CHECK ON
OR        M1902F	// DRY RUN
OUT       M1007A	// L_1st MANDREL DIE VACUUM CHECK ON
// ======================== CONDITION SETTING ==========================
; L91
LOAD      M10010	// 01_AU¥ì¢¯ AUAc & CC¢¥o E¢çAI
AND       M10190	// L_1st MAND PICKER ENABLE
AND NOT   M10180	// L_1st MAND AU¨ú¡À¢¯I¡¤a
AND       M04030	// L_1-1 ROT R IDLE POS
AND       M04050	// L_1st ROT Y 1st POS
AND       P00020	// L_1st TOP CLAMP UP
AND       T1016	// L_1st DIE ALIGN BACKWARD
AND       T1018	// L_1st DIE FPCB ALIGN BACKWARD
AND       P00025	// L_1st ROTATE MANDREL BACKWARD
AND       P00110	// L_1st DIE VACUUM EJECTOR ON
AND       M1007A	// L_1st MANDREL DIE VACUUM CHECK ON
OUT       M10030	// STEP A¢Ò¡ÆC1
// output comment: 01_AU¥ì¢¯ AUAc & CC¢¥o E¢çAI
; L92
LOAD      P00022	// L_1st DIE ALIGN FORWARD
AND       M04030	// L_1-1 ROT R IDLE POS
AND       M04050	// L_1st ROT Y 1st POS
AND       P00020	// L_1st TOP CLAMP UP
AND       T1018	// L_1st DIE FPCB ALIGN BACKWARD
AND       P00025	// L_1st ROTATE MANDREL BACKWARD
AND       P00110	// L_1st DIE VACUUM EJECTOR ON
OUT       M10031	// STEP A¢Ò¡ÆC2
// output comment: 01_AU¥ì¢¯ ¨úo¢ÒoAI AuA©ª
; L93
LOAD      P00023	// L_1st DIE FPCB ALIGN FORWARD
AND       P00020	// L_1st TOP CLAMP UP
AND       P00022	// L_1st DIE ALIGN FORWARD
AND       M04030	// L_1-1 ROT R IDLE POS
AND       M04050	// L_1st ROT Y 1st POS
AND       P00025	// L_1st ROTATE MANDREL BACKWARD
AND       P00110	// L_1st DIE VACUUM EJECTOR ON
OUT       M10032	// STEP A¢Ò¡ÆC3
// output comment: 01_AU¥ì¢¯ FPCB ¨úo¢ÒoAI AuA©ª
; L94
LOAD      P00021	// L_1st TOP CLAMP DONW
AND       M04030	// L_1-1 ROT R IDLE POS
AND       M04050	// L_1st ROT Y 1st POS
AND       P00022	// L_1st DIE ALIGN FORWARD
AND       P00023	// L_1st DIE FPCB ALIGN FORWARD
AND       P00025	// L_1st ROTATE MANDREL BACKWARD
AND       P00110	// L_1st DIE VACUUM EJECTOR ON
OUT       M10033	// STEP A¢Ò¡ÆC4
// output comment: 01_AU¥ì¢¯ A¡þ¡¤¡ÍCA Z CI¡Æ¡©->

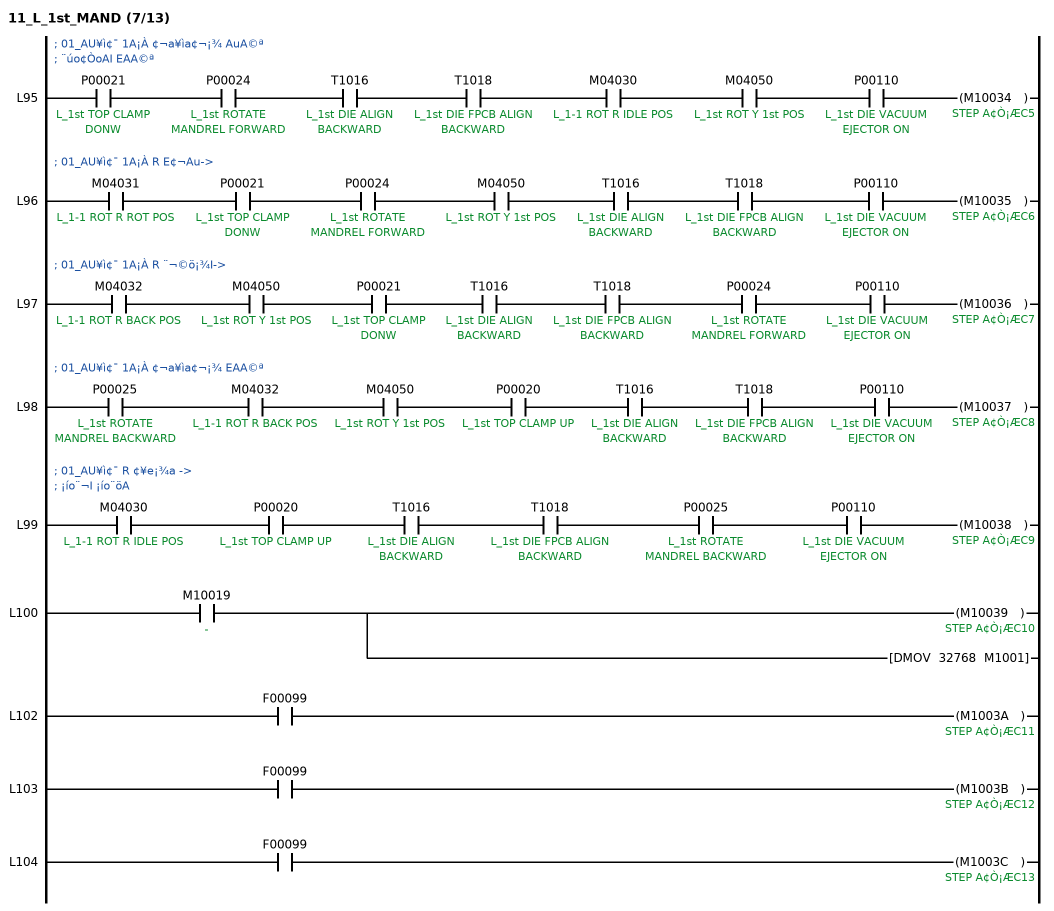
; L95
LOAD      P00021	// L_1st TOP CLAMP DONW
AND       P00024	// L_1st ROTATE MANDREL FORWARD
AND       T1016	// L_1st DIE ALIGN BACKWARD
AND       T1018	// L_1st DIE FPCB ALIGN BACKWARD
AND       M04030	// L_1-1 ROT R IDLE POS
AND       M04050	// L_1st ROT Y 1st POS
AND       P00110	// L_1st DIE VACUUM EJECTOR ON
OUT       M10034	// STEP A¢Ò¡ÆC5
// output comment: 01_AU¥ì¢¯ 1A¡À ¢¬a¥ìa¢¬¡¾ AuA©ª ¨úo¢ÒoAI EAA©ª
; L96
LOAD      M04031	// L_1-1 ROT R ROT POS
AND       P00021	// L_1st TOP CLAMP DONW
AND       P00024	// L_1st ROTATE MANDREL FORWARD
AND       M04050	// L_1st ROT Y 1st POS
AND       T1016	// L_1st DIE ALIGN BACKWARD
AND       T1018	// L_1st DIE FPCB ALIGN BACKWARD
AND       P00110	// L_1st DIE VACUUM EJECTOR ON
OUT       M10035	// STEP A¢Ò¡ÆC6
// output comment: 01_AU¥ì¢¯ 1A¡À R E¢¬Au->
; L97
LOAD      M04032	// L_1-1 ROT R BACK POS
AND       M04050	// L_1st ROT Y 1st POS
AND       P00021	// L_1st TOP CLAMP DONW
AND       T1016	// L_1st DIE ALIGN BACKWARD
AND       T1018	// L_1st DIE FPCB ALIGN BACKWARD
AND       P00024	// L_1st ROTATE MANDREL FORWARD
AND       P00110	// L_1st DIE VACUUM EJECTOR ON
OUT       M10036	// STEP A¢Ò¡ÆC7
// output comment: 01_AU¥ì¢¯ 1A¡À R ¨¬©ö¡¾I->
; L98
LOAD      P00025	// L_1st ROTATE MANDREL BACKWARD
AND       M04032	// L_1-1 ROT R BACK POS
AND       M04050	// L_1st ROT Y 1st POS
AND       P00020	// L_1st TOP CLAMP UP
AND       T1016	// L_1st DIE ALIGN BACKWARD
AND       T1018	// L_1st DIE FPCB ALIGN BACKWARD
AND       P00110	// L_1st DIE VACUUM EJECTOR ON
OUT       M10037	// STEP A¢Ò¡ÆC8
// output comment: 01_AU¥ì¢¯ 1A¡À ¢¬a¥ìa¢¬¡¾ EAA©ª
; L99
LOAD      M04030	// L_1-1 ROT R IDLE POS
AND       P00020	// L_1st TOP CLAMP UP
AND       T1016	// L_1st DIE ALIGN BACKWARD
AND       T1018	// L_1st DIE FPCB ALIGN BACKWARD
AND       P00025	// L_1st ROTATE MANDREL BACKWARD
AND       P00110	// L_1st DIE VACUUM EJECTOR ON
OUT       M10038	// STEP A¢Ò¡ÆC9
// output comment: 01_AU¥ì¢¯ R ¢¥e¡¾a -> ¡ío¨¬I ¡ío¨öA
; L100
LOAD      M10019	// -
OUT       M10039	// STEP A¢Ò¡ÆC10
DMOV      32768 M1001
; L102
LOAD      F00099
OUT       M1003A	// STEP A¢Ò¡ÆC11
; L103
LOAD      F00099
OUT       M1003B	// STEP A¢Ò¡ÆC12
; L104
LOAD      F00099
OUT       M1003C	// STEP A¢Ò¡ÆC13

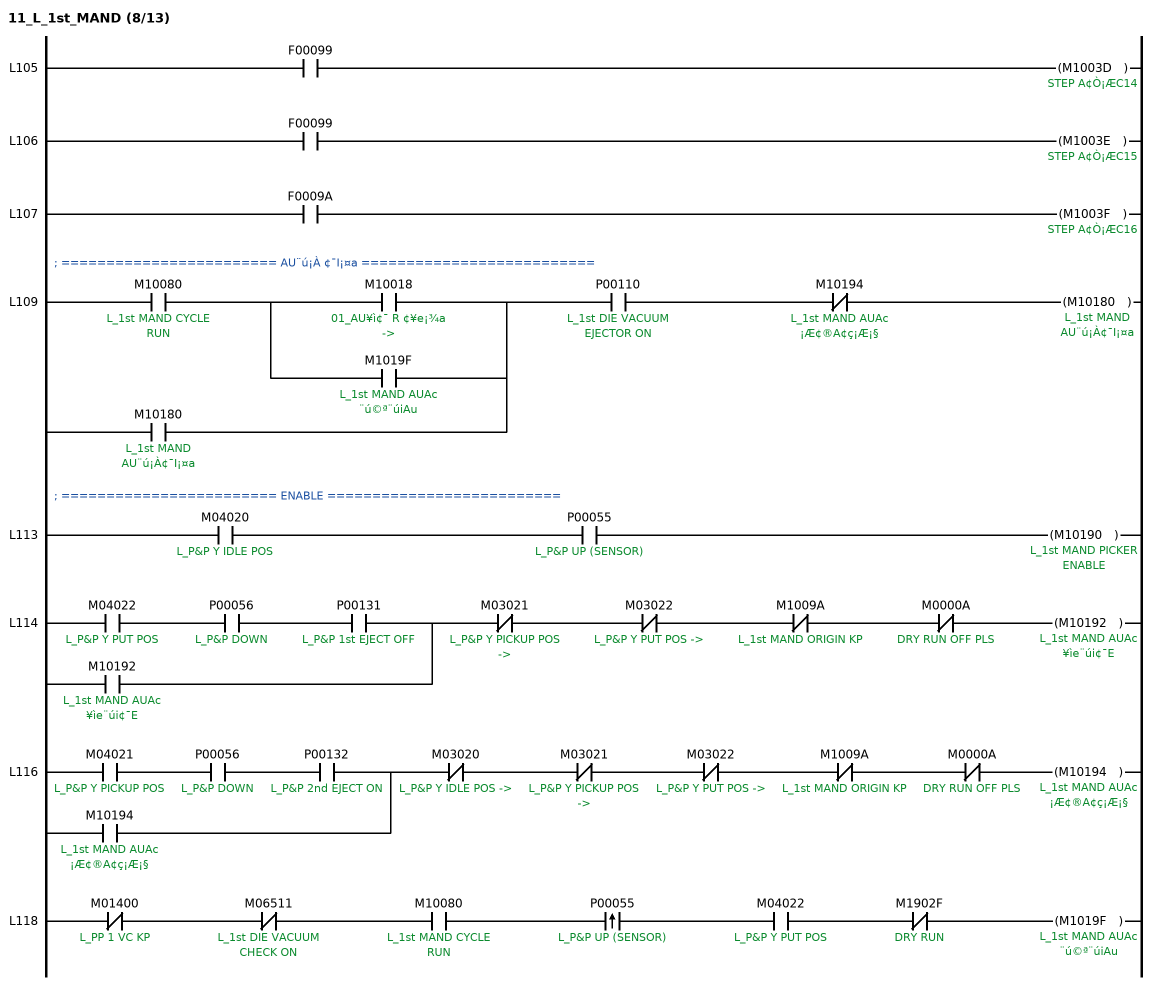
; L105
LOAD      F00099
OUT       M1003D	// STEP A¢Ò¡ÆC14
; L106
LOAD      F00099
OUT       M1003E	// STEP A¢Ò¡ÆC15
; L107
LOAD      F0009A
OUT       M1003F	// STEP A¢Ò¡ÆC16
// ======================== AU¨ú¡À ¢¯I¡¤a ==========================
; L109
LOAD      M10080	// L_1st MAND CYCLE RUN
LOAD      M10018	// 01_AU¥ì¢¯ R ¢¥e¡¾a ->
OR        M1019F	// L_1st MAND AUAc ¨ú©ª¨úiAu
AND LOAD
OR        M10180	// L_1st MAND AU¨ú¡À¢¯I¡¤a
AND       P00110	// L_1st DIE VACUUM EJECTOR ON
AND NOT   M10194	// L_1st MAND AUAc ¡Æ¢®A¢ç¡Æ¡§
OUT       M10180	// L_1st MAND AU¨ú¡À¢¯I¡¤a
// ======================== ENABLE ==========================
; L113
LOAD      M04020	// L_P&P Y IDLE POS
AND       P00055	// L_P&P UP (SENSOR)
OUT       M10190	// L_1st MAND PICKER ENABLE
; L114
LOAD      M04022	// L_P&P Y PUT POS
AND       P00056	// L_P&P DOWN
AND       P00131	// L_P&P 1st EJECT OFF
OR        M10192	// L_1st MAND AUAc ¥ìe¨úi¢¯E
AND NOT   M03021	// L_P&P Y PICKUP POS ->
AND NOT   M03022	// L_P&P Y PUT POS ->
AND NOT   M1009A	// L_1st MAND ORIGIN KP
AND NOT   M0000A	// DRY RUN OFF PLS
OUT       M10192	// L_1st MAND AUAc ¥ìe¨úi¢¯E
; L116
LOAD      M04021	// L_P&P Y PICKUP POS
AND       P00056	// L_P&P DOWN
AND       P00132	// L_P&P 2nd EJECT ON
OR        M10194	// L_1st MAND AUAc ¡Æ¢®A¢ç¡Æ¡§
AND NOT   M03020	// L_P&P Y IDLE POS ->
AND NOT   M03021	// L_P&P Y PICKUP POS ->
AND NOT   M03022	// L_P&P Y PUT POS ->
AND NOT   M1009A	// L_1st MAND ORIGIN KP
AND NOT   M0000A	// DRY RUN OFF PLS
OUT       M10194	// L_1st MAND AUAc ¡Æ¢®A¢ç¡Æ¡§
; L118
LOAD NOT  M01400	// L_PP 1 VC KP
AND NOT   M06511	// L_1st DIE VACUUM CHECK ON
AND       M10080	// L_1st MAND CYCLE RUN
ANDP      P00055	// L_P&P UP (SENSOR)
AND       M04022	// L_P&P Y PUT POS
AND NOT   M1902F	// DRY RUN
OUT       M1019F	// L_1st MAND AUAc ¨ú©ª¨úiAu

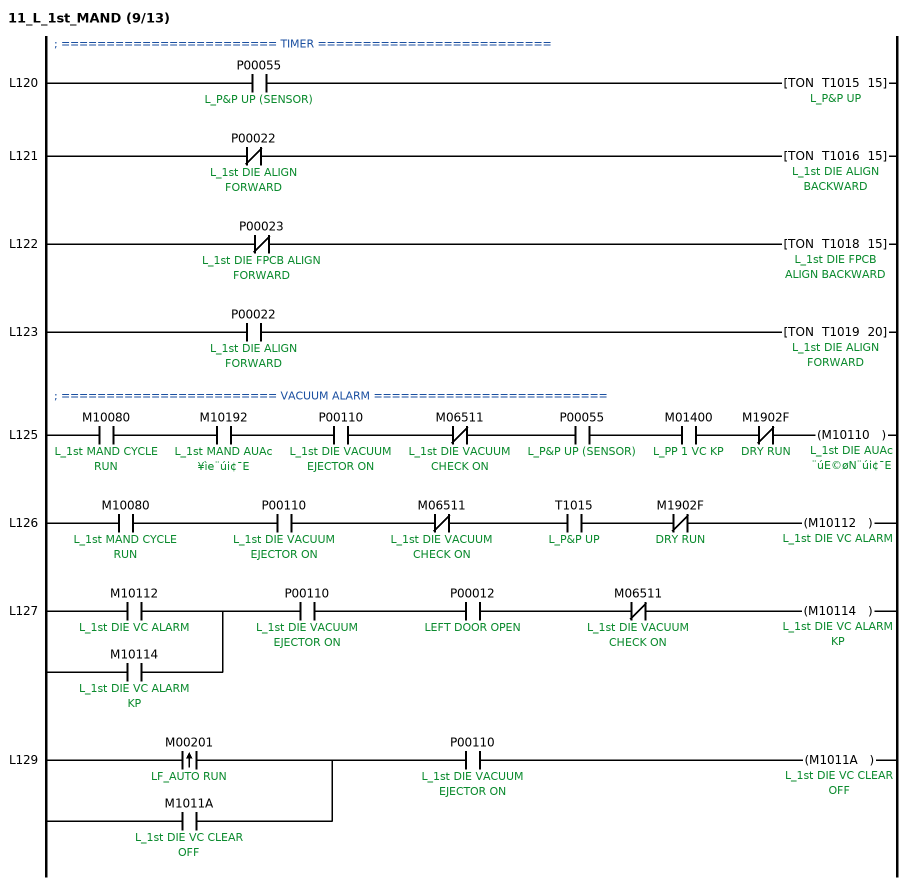
// ======================== TIMER ==========================
; L120
LOAD      P00055	// L_P&P UP (SENSOR)
TON       T1015 15	// L_P&P UP
; L121
LOAD NOT  P00022	// L_1st DIE ALIGN FORWARD
TON       T1016 15	// L_1st DIE ALIGN BACKWARD
; L122
LOAD NOT  P00023	// L_1st DIE FPCB ALIGN FORWARD
TON       T1018 15	// L_1st DIE FPCB ALIGN BACKWARD
; L123
LOAD      P00022	// L_1st DIE ALIGN FORWARD
TON       T1019 20	// L_1st DIE ALIGN FORWARD
// ======================== VACUUM ALARM ==========================
; L125
LOAD      M10080	// L_1st MAND CYCLE RUN
AND       M10192	// L_1st MAND AUAc ¥ìe¨úi¢¯E
AND       P00110	// L_1st DIE VACUUM EJECTOR ON
AND NOT   M06511	// L_1st DIE VACUUM CHECK ON
AND       P00055	// L_P&P UP (SENSOR)
AND       M01400	// L_PP 1 VC KP
AND NOT   M1902F	// DRY RUN
OUT       M10110	// L_1st DIE AUAc ¨úE©øN¨úi¢¯E
; L126
LOAD      M10080	// L_1st MAND CYCLE RUN
AND       P00110	// L_1st DIE VACUUM EJECTOR ON
AND NOT   M06511	// L_1st DIE VACUUM CHECK ON
AND       T1015	// L_P&P UP
AND NOT   M1902F	// DRY RUN
OUT       M10112	// L_1st DIE VC ALARM
; L127
LOAD      M10112	// L_1st DIE VC ALARM
OR        M10114	// L_1st DIE VC ALARM KP
AND       P00110	// L_1st DIE VACUUM EJECTOR ON
AND       P00012	// LEFT DOOR OPEN
AND NOT   M06511	// L_1st DIE VACUUM CHECK ON
OUT       M10114	// L_1st DIE VC ALARM KP
; L129
LOADP     M00201	// LF_AUTO RUN
OR        M1011A	// L_1st DIE VC CLEAR OFF
AND       P00110	// L_1st DIE VACUUM EJECTOR ON
OUT       M1011A	// L_1st DIE VC CLEAR OFF

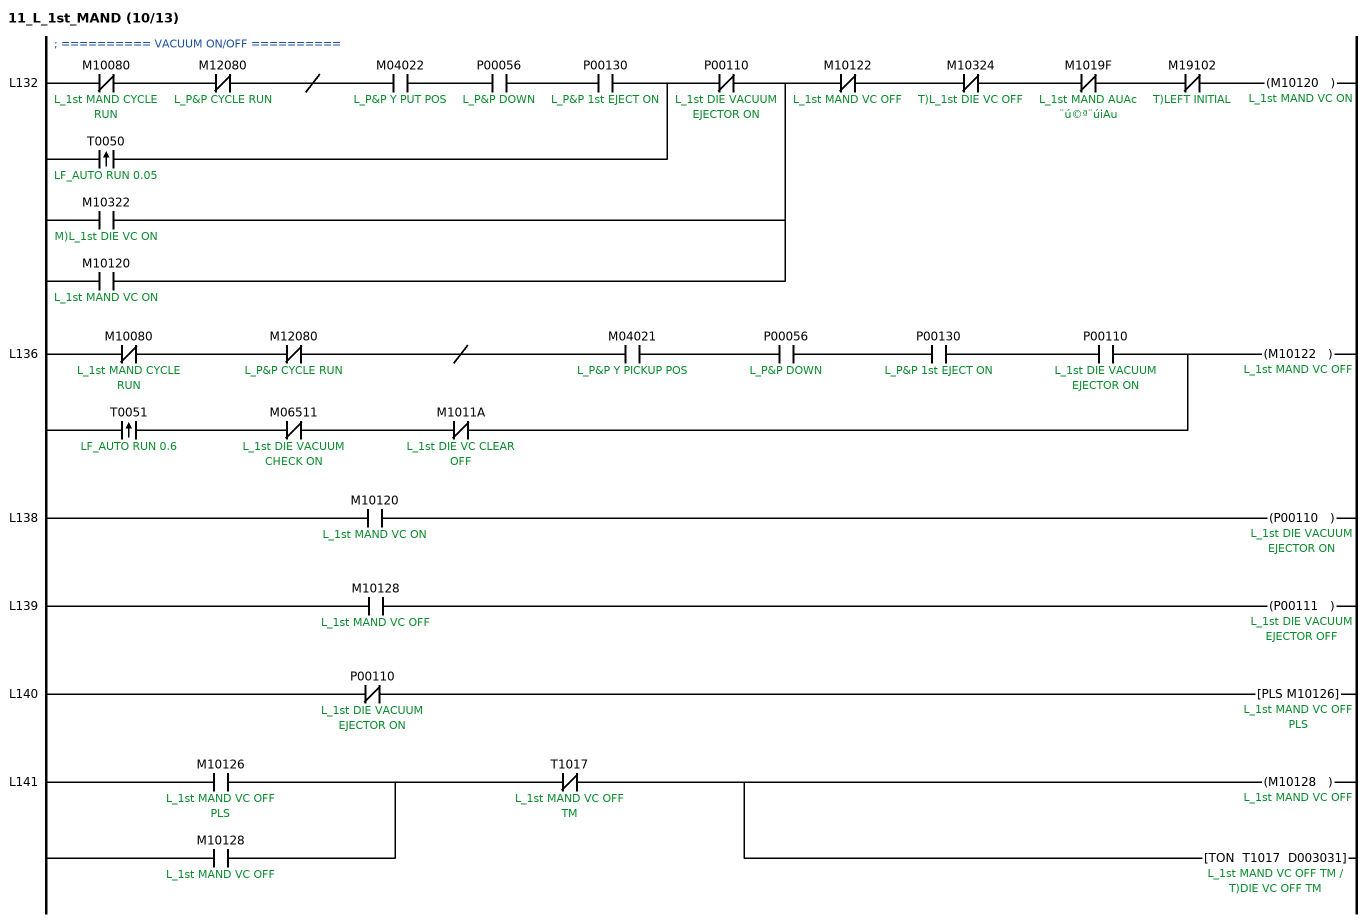
// ========== VACUUM ON/OFF ==========
; L132
LOAD NOT  M10080	// L_1st MAND CYCLE RUN
AND NOT   M12080	// L_P&P CYCLE RUN
NOT
AND       M04022	// L_P&P Y PUT POS
AND       P00056	// L_P&P DOWN
AND       P00130	// L_P&P 1st EJECT ON
ORP       T0050	// LF_AUTO RUN 0.05
AND NOT   P00110	// L_1st DIE VACUUM EJECTOR ON
OR        M10322	// M)L_1st DIE VC ON
OR        M10120	// L_1st MAND VC ON
AND NOT   M10122	// L_1st MAND VC OFF
AND NOT   M10324	// T)L_1st DIE VC OFF
AND NOT   M1019F	// L_1st MAND AUAc ¨ú©ª¨úiAu
AND NOT   M19102	// T)LEFT INITIAL
OUT       M10120	// L_1st MAND VC ON
; L136
LOAD NOT  M10080	// L_1st MAND CYCLE RUN
AND NOT   M12080	// L_P&P CYCLE RUN
NOT
AND       M04021	// L_P&P Y PICKUP POS
AND       P00056	// L_P&P DOWN
AND       P00130	// L_P&P 1st EJECT ON
AND       P00110	// L_1st DIE VACUUM EJECTOR ON
LOADP     T0051	// LF_AUTO RUN 0.6
AND NOT   M06511	// L_1st DIE VACUUM CHECK ON
AND NOT   M1011A	// L_1st DIE VC CLEAR OFF
OR LOAD
OUT       M10122	// L_1st MAND VC OFF
; L138
LOAD      M10120	// L_1st MAND VC ON
OUT       P00110	// L_1st DIE VACUUM EJECTOR ON
; L139
LOAD      M10128	// L_1st MAND VC OFF
OUT       P00111	// L_1st DIE VACUUM EJECTOR OFF
; L140
LOAD NOT  P00110	// L_1st DIE VACUUM EJECTOR ON
OUTP      M10126	// L_1st MAND VC OFF PLS
; L141
LOAD      M10126	// L_1st MAND VC OFF PLS
OR        M10128	// L_1st MAND VC OFF
AND NOT   T1017	// L_1st MAND VC OFF TM
OUT       M10128	// L_1st MAND VC OFF
TON       T1017 D003031	// L_1st MAND VC OFF TM / T)DIE VC OFF TM

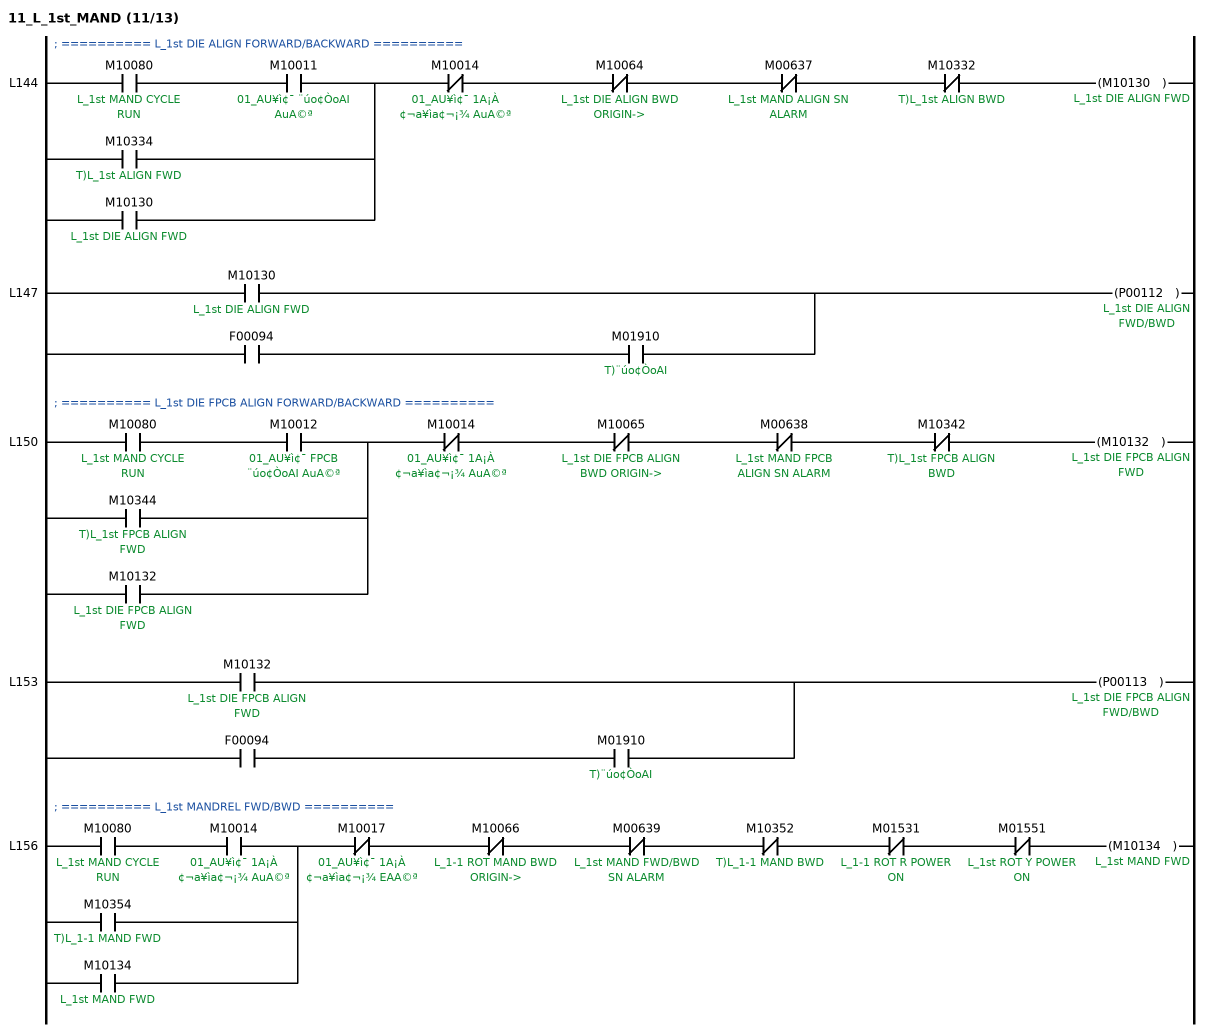
// ========== L_1st DIE ALIGN FORWARD/BACKWARD ==========
; L144
LOAD      M10080	// L_1st MAND CYCLE RUN
AND       M10011	// 01_AU¥ì¢¯ ¨úo¢ÒoAI AuA©ª
OR        M10334	// T)L_1st ALIGN FWD
OR        M10130	// L_1st DIE ALIGN FWD
AND NOT   M10014	// 01_AU¥ì¢¯ 1A¡À ¢¬a¥ìa¢¬¡¾ AuA©ª
AND NOT   M10064	// L_1st DIE ALIGN BWD ORIGIN->
AND NOT   M00637	// L_1st MAND ALIGN SN ALARM
AND NOT   M10332	// T)L_1st ALIGN BWD
OUT       M10130	// L_1st DIE ALIGN FWD
; L147
LOAD      M10130	// L_1st DIE ALIGN FWD
LOAD      F00094
AND       M01910	// T)¨úo¢ÒoAI
OR LOAD
OUT       P00112	// L_1st DIE ALIGN FWD/BWD
// ========== L_1st DIE FPCB ALIGN FORWARD/BACKWARD ==========
; L150
LOAD      M10080	// L_1st MAND CYCLE RUN
AND       M10012	// 01_AU¥ì¢¯ FPCB ¨úo¢ÒoAI AuA©ª
OR        M10344	// T)L_1st FPCB ALIGN FWD
OR        M10132	// L_1st DIE FPCB ALIGN FWD
AND NOT   M10014	// 01_AU¥ì¢¯ 1A¡À ¢¬a¥ìa¢¬¡¾ AuA©ª
AND NOT   M10065	// L_1st DIE FPCB ALIGN BWD ORIGIN->
AND NOT   M00638	// L_1st MAND FPCB ALIGN SN ALARM
AND NOT   M10342	// T)L_1st FPCB ALIGN BWD
OUT       M10132	// L_1st DIE FPCB ALIGN FWD
; L153
LOAD      M10132	// L_1st DIE FPCB ALIGN FWD
LOAD      F00094
AND       M01910	// T)¨úo¢ÒoAI
OR LOAD
OUT       P00113	// L_1st DIE FPCB ALIGN FWD/BWD
// ========== L_1st MANDREL FWD/BWD ==========
; L156
LOAD      M10080	// L_1st MAND CYCLE RUN
AND       M10014	// 01_AU¥ì¢¯ 1A¡À ¢¬a¥ìa¢¬¡¾ AuA©ª
OR        M10354	// T)L_1-1 MAND FWD
OR        M10134	// L_1st MAND FWD
AND NOT   M10017	// 01_AU¥ì¢¯ 1A¡À ¢¬a¥ìa¢¬¡¾ EAA©ª
AND NOT   M10066	// L_1-1 ROT MAND BWD ORIGIN->
AND NOT   M00639	// L_1st MAND FWD/BWD SN ALARM
AND NOT   M10352	// T)L_1-1 MAND BWD
AND NOT   M01531	// L_1-1 ROT R POWER ON
AND NOT   M01551	// L_1st ROT Y POWER ON
OUT       M10134	// L_1st MAND FWD

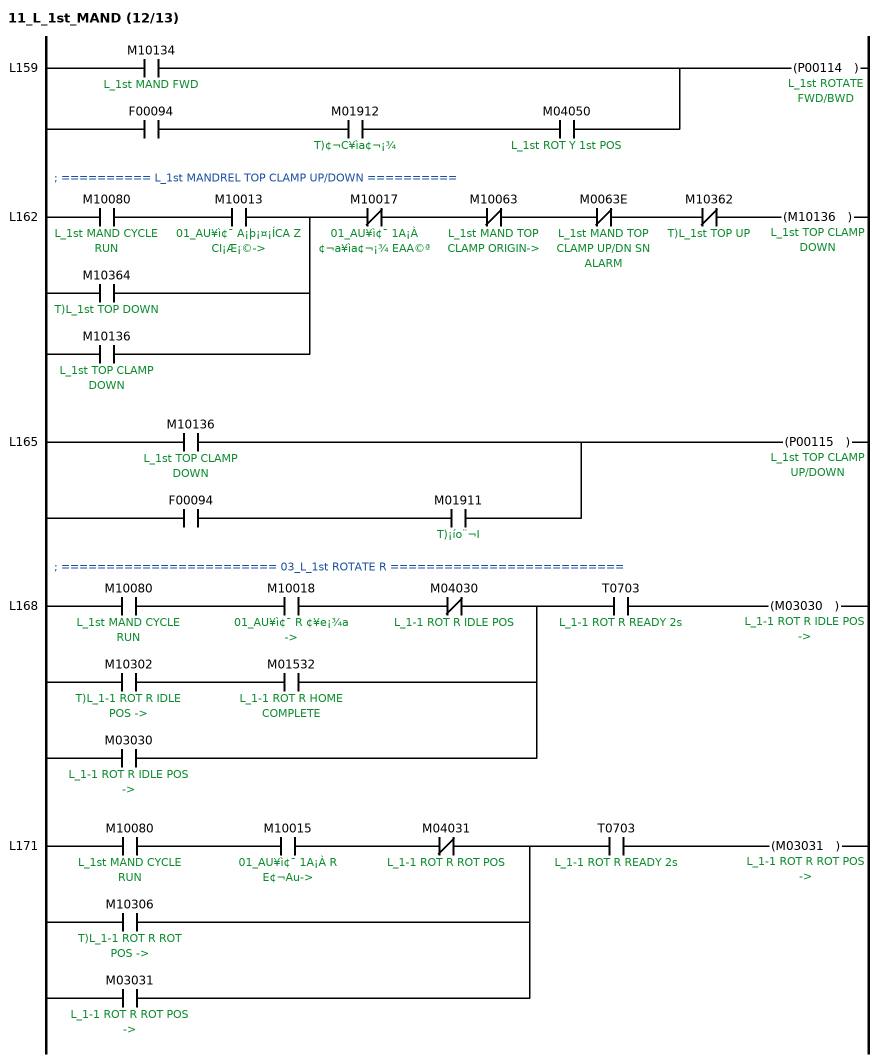
; L159
LOAD      M10134	// L_1st MAND FWD
LOAD      F00094
AND       M01912	// T)¢¬C¥ìa¢¬¡¾
AND       M04050	// L_1st ROT Y 1st POS
OR LOAD
OUT       P00114	// L_1st ROTATE FWD/BWD
// ========== L_1st MANDREL TOP CLAMP UP/DOWN ==========
; L162
LOAD      M10080	// L_1st MAND CYCLE RUN
AND       M10013	// 01_AU¥ì¢¯ A¡þ¡¤¡ÍCA Z CI¡Æ¡©->
OR        M10364	// T)L_1st TOP DOWN
OR        M10136	// L_1st TOP CLAMP DOWN
AND NOT   M10017	// 01_AU¥ì¢¯ 1A¡À ¢¬a¥ìa¢¬¡¾ EAA©ª
AND NOT   M10063	// L_1st MAND TOP CLAMP ORIGIN->
AND NOT   M0063E	// L_1st MAND TOP CLAMP UP/DN SN ALARM
AND NOT   M10362	// T)L_1st TOP UP
OUT       M10136	// L_1st TOP CLAMP DOWN
; L165
LOAD      M10136	// L_1st TOP CLAMP DOWN
LOAD      F00094
AND       M01911	// T)¡ío¨¬I
OR LOAD
OUT       P00115	// L_1st TOP CLAMP UP/DOWN
// ======================== 03_L_1st ROTATE R ==========================
; L168
LOAD      M10080	// L_1st MAND CYCLE RUN
AND       M10018	// 01_AU¥ì¢¯ R ¢¥e¡¾a ->
AND NOT   M04030	// L_1-1 ROT R IDLE POS
LOAD      M10302	// T)L_1-1 ROT R IDLE POS ->
AND       M01532	// L_1-1 ROT R HOME COMPLETE
OR LOAD
OR        M03030	// L_1-1 ROT R IDLE POS ->
AND       T0703	// L_1-1 ROT R READY 2s
OUT       M03030	// L_1-1 ROT R IDLE POS ->
; L171
LOAD      M10080	// L_1st MAND CYCLE RUN
AND       M10015	// 01_AU¥ì¢¯ 1A¡À R E¢¬Au->
AND NOT   M04031	// L_1-1 ROT R ROT POS
OR        M10306	// T)L_1-1 ROT R ROT POS ->
OR        M03031	// L_1-1 ROT R ROT POS ->
AND       T0703	// L_1-1 ROT R READY 2s
OUT       M03031	// L_1-1 ROT R ROT POS ->

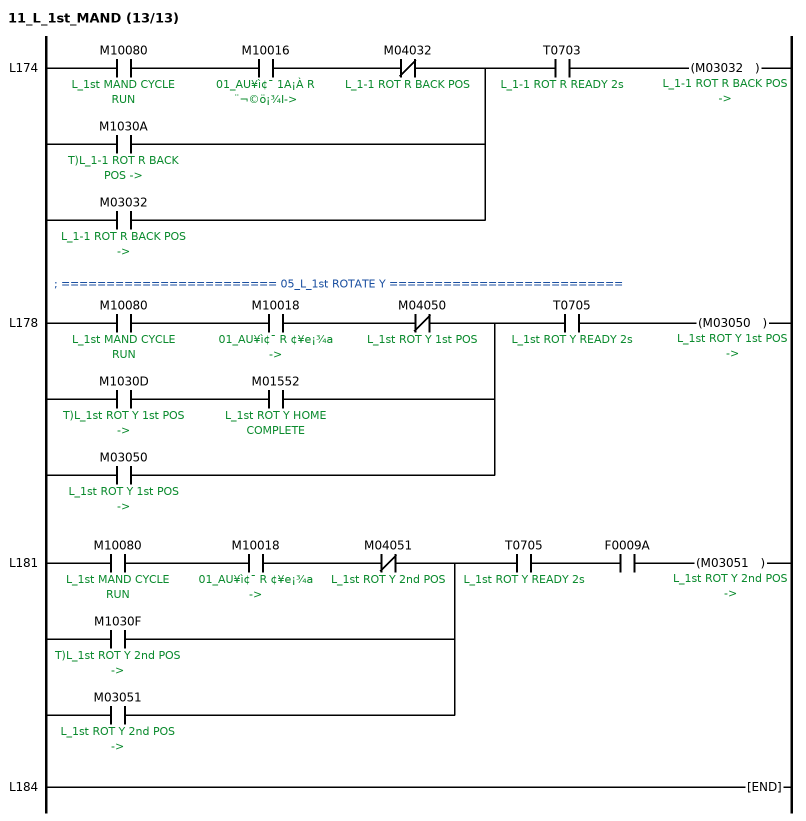
; L174
LOAD      M10080	// L_1st MAND CYCLE RUN
AND       M10016	// 01_AU¥ì¢¯ 1A¡À R ¨¬©ö¡¾I->
AND NOT   M04032	// L_1-1 ROT R BACK POS
OR        M1030A	// T)L_1-1 ROT R BACK POS ->
OR        M03032	// L_1-1 ROT R BACK POS ->
AND       T0703	// L_1-1 ROT R READY 2s
OUT       M03032	// L_1-1 ROT R BACK POS ->
// ======================== 05_L_1st ROTATE Y ==========================
; L178
LOAD      M10080	// L_1st MAND CYCLE RUN
AND       M10018	// 01_AU¥ì¢¯ R ¢¥e¡¾a ->
AND NOT   M04050	// L_1st ROT Y 1st POS
LOAD      M1030D	// T)L_1st ROT Y 1st POS ->
AND       M01552	// L_1st ROT Y HOME COMPLETE
OR LOAD
OR        M03050	// L_1st ROT Y 1st POS ->
AND       T0705	// L_1st ROT Y READY 2s
OUT       M03050	// L_1st ROT Y 1st POS ->
; L181
LOAD      M10080	// L_1st MAND CYCLE RUN
AND       M10018	// 01_AU¥ì¢¯ R ¢¥e¡¾a ->
AND NOT   M04051	// L_1st ROT Y 2nd POS
OR        M1030F	// T)L_1st ROT Y 2nd POS ->
OR        M03051	// L_1st ROT Y 2nd POS ->
AND       T0705	// L_1st ROT Y READY 2s
AND       F0009A
OUT       M03051	// L_1st ROT Y 2nd POS ->
; L184
END

PROGRAM 12_L_2nd_MAND (task: ¨ö¨¬A¥ì CA¡¤I¡¾¡¿¡¤¡Í)

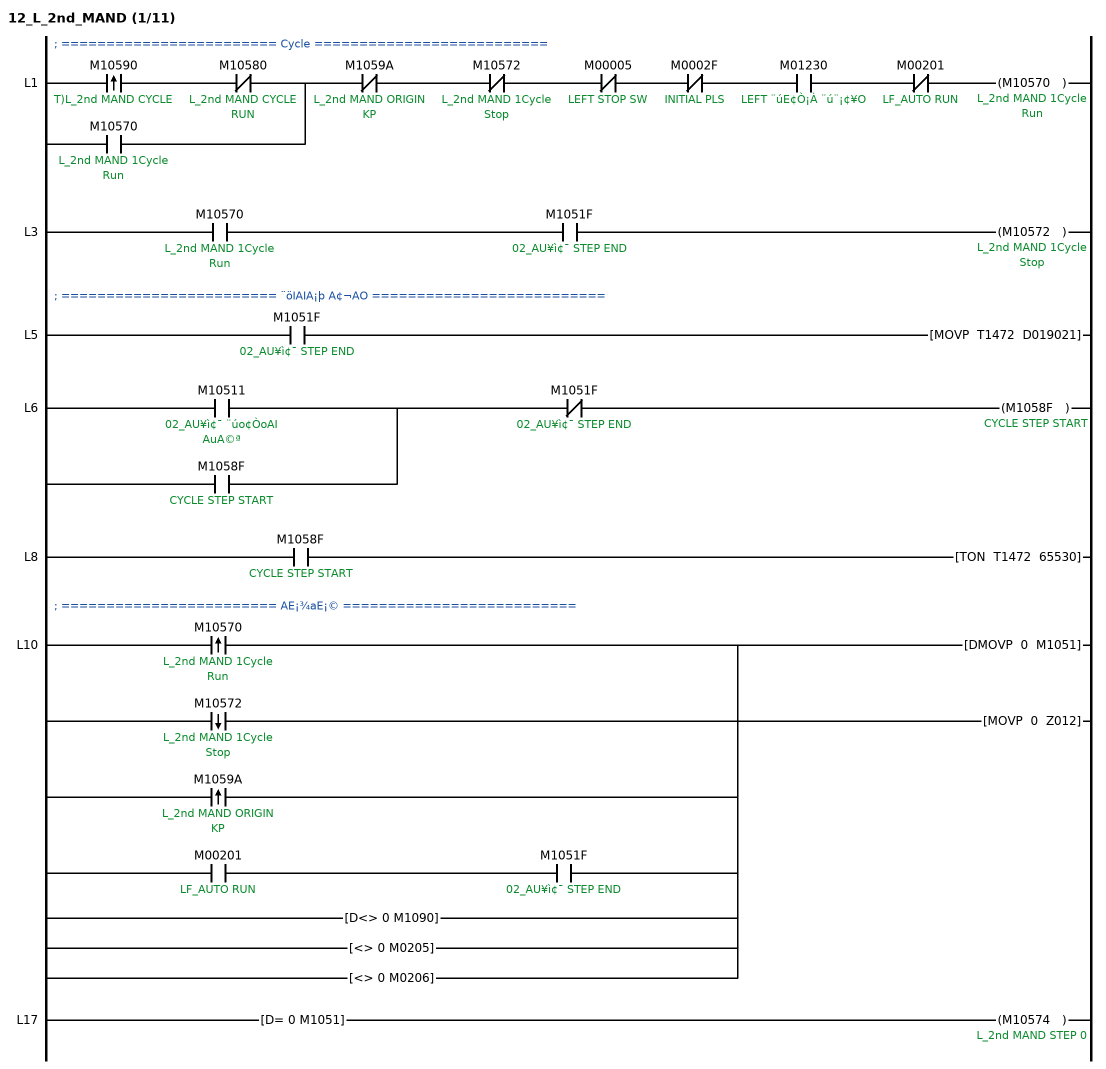
// ======================== Cycle ==========================
; L1
LOADP     M10590	// T)L_2nd MAND CYCLE
AND NOT   M10580	// L_2nd MAND CYCLE RUN
OR        M10570	// L_2nd MAND 1Cycle Run
AND NOT   M1059A	// L_2nd MAND ORIGIN KP
AND NOT   M10572	// L_2nd MAND 1Cycle Stop
AND NOT   M00005	// LEFT STOP SW
AND NOT   M0002F	// INITIAL PLS
AND       M01230	// LEFT ¨úE¢Ò¡À ¨ú¨¡¢¥O
AND NOT   M00201	// LF_AUTO RUN
OUT       M10570	// L_2nd MAND 1Cycle Run
; L3
LOAD      M10570	// L_2nd MAND 1Cycle Run
AND       M1051F	// 02_AU¥ì¢¯ STEP END
OUT       M10572	// L_2nd MAND 1Cycle Stop
// ======================== ¨öIAIA¡þ A¢¬AO ==========================
; L5
LOAD      M1051F	// 02_AU¥ì¢¯ STEP END
MOVP      T1472 D019021
; L6
LOAD      M10511	// 02_AU¥ì¢¯ ¨úo¢ÒoAI AuA©ª
OR        M1058F	// CYCLE STEP START
AND NOT   M1051F	// 02_AU¥ì¢¯ STEP END
OUT       M1058F	// CYCLE STEP START
; L8
LOAD      M1058F	// CYCLE STEP START
TON       T1472 65530
// ======================== AE¡¾aE¡© ==========================
; L10
LOADP     M10570	// L_2nd MAND 1Cycle Run
ORN       M10572	// L_2nd MAND 1Cycle Stop
ORP       M1059A	// L_2nd MAND ORIGIN KP
LOAD      M00201	// LF_AUTO RUN
AND       M1051F	// 02_AU¥ì¢¯ STEP END
OR LOAD
ORD<>     0 M1090
OR<>      0 M0205
OR<>      0 M0206
DMOVP     0 M1051
MOVP      0 Z012
; L17
LOADD=    0 M1051
OUT       M10574	// L_2nd MAND STEP 0

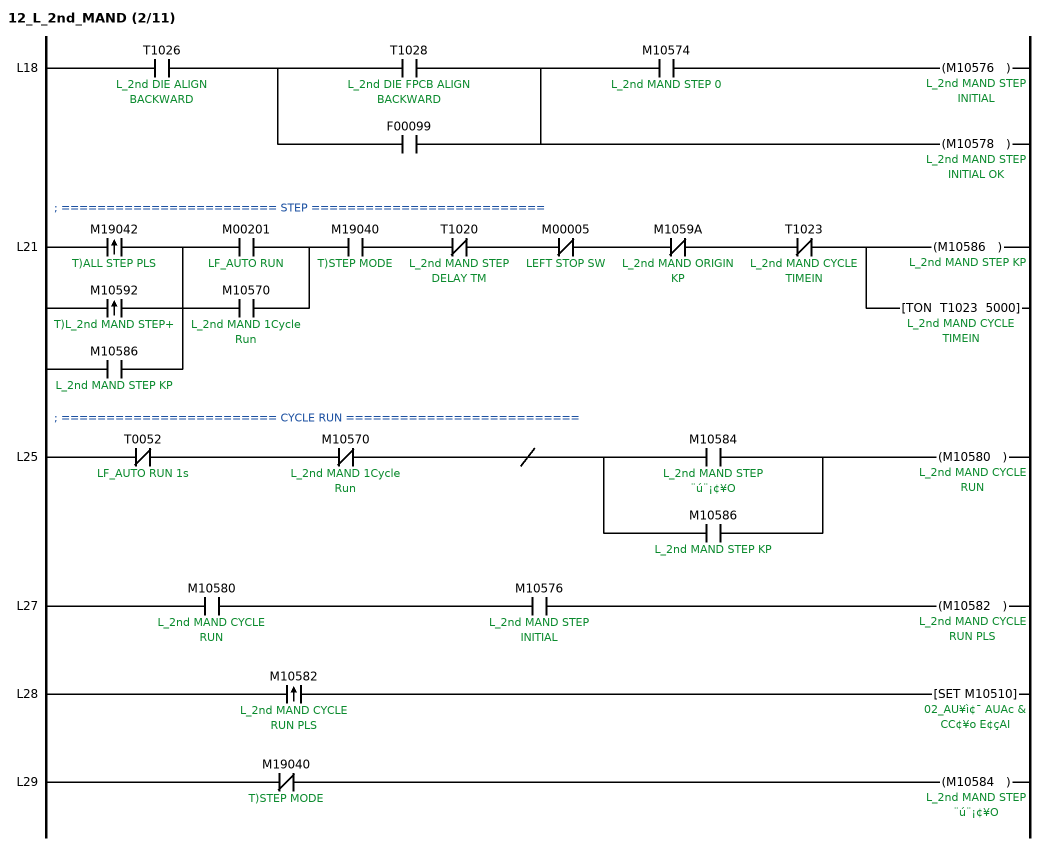
; L18
LOAD      T1026	// L_2nd DIE ALIGN BACKWARD
LOAD      T1028	// L_2nd DIE FPCB ALIGN BACKWARD
OR        F00099
AND LOAD
MPUSH
AND       M10574	// L_2nd MAND STEP 0
OUT       M10576	// L_2nd MAND STEP INITIAL
MPOP
OUT       M10578	// L_2nd MAND STEP INITIAL OK
// ======================== STEP ==========================
; L21
LOADP     M19042	// T)ALL STEP PLS
ORP       M10592	// T)L_2nd MAND STEP+
OR        M10586	// L_2nd MAND STEP KP
LOAD      M00201	// LF_AUTO RUN
OR        M10570	// L_2nd MAND 1Cycle Run
AND LOAD
AND       M19040	// T)STEP MODE
AND NOT   T1020	// L_2nd MAND STEP DELAY TM
AND NOT   M00005	// LEFT STOP SW
AND NOT   M1059A	// L_2nd MAND ORIGIN KP
AND NOT   T1023	// L_2nd MAND CYCLE TIMEIN
OUT       M10586	// L_2nd MAND STEP KP
TON       T1023 5000	// L_2nd MAND CYCLE TIMEIN
// ======================== CYCLE RUN ==========================
; L25
LOAD NOT  T0052	// LF_AUTO RUN 1s
AND NOT   M10570	// L_2nd MAND 1Cycle Run
NOT
LOAD      M10584	// L_2nd MAND STEP ¨ú¨¡¢¥O
OR        M10586	// L_2nd MAND STEP KP
AND LOAD
OUT       M10580	// L_2nd MAND CYCLE RUN
; L27
LOAD      M10580	// L_2nd MAND CYCLE RUN
AND       M10576	// L_2nd MAND STEP INITIAL
OUT       M10582	// L_2nd MAND CYCLE RUN PLS
; L28
LOADP     M10582	// L_2nd MAND CYCLE RUN PLS
SET       M10510	// 02_AU¥ì¢¯ AUAc & CC¢¥o E¢çAI
; L29
LOAD NOT  M19040	// T)STEP MODE
OUT       M10584	// L_2nd MAND STEP ¨ú¨¡¢¥O

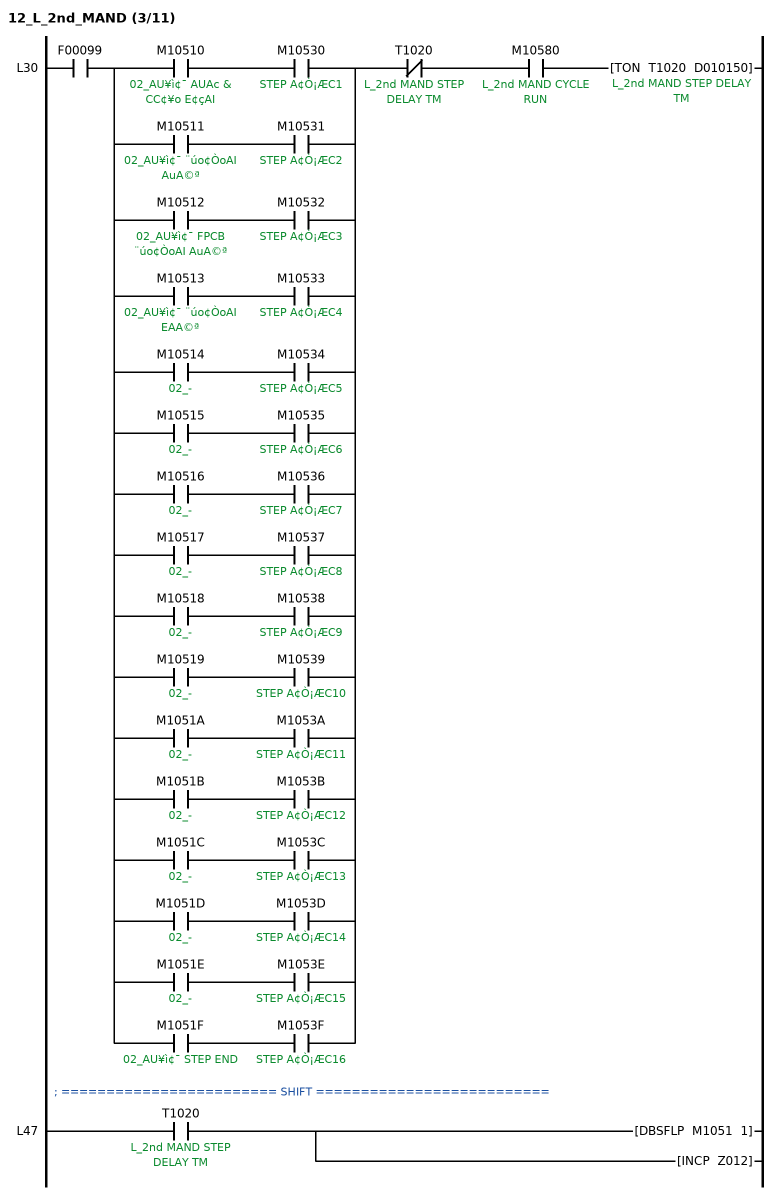
; L30
LOAD      F00099
LOAD      M10510	// 02_AU¥ì¢¯ AUAc & CC¢¥o E¢çAI
AND       M10530	// STEP A¢Ò¡ÆC1
LOAD      M10511	// 02_AU¥ì¢¯ ¨úo¢ÒoAI AuA©ª
AND       M10531	// STEP A¢Ò¡ÆC2
OR LOAD
LOAD      M10512	// 02_AU¥ì¢¯ FPCB ¨úo¢ÒoAI AuA©ª
AND       M10532	// STEP A¢Ò¡ÆC3
OR LOAD
LOAD      M10513	// 02_AU¥ì¢¯ ¨úo¢ÒoAI EAA©ª
AND       M10533	// STEP A¢Ò¡ÆC4
OR LOAD
LOAD      M10514	// 02_-
AND       M10534	// STEP A¢Ò¡ÆC5
OR LOAD
LOAD      M10515	// 02_-
AND       M10535	// STEP A¢Ò¡ÆC6
OR LOAD
LOAD      M10516	// 02_-
AND       M10536	// STEP A¢Ò¡ÆC7
OR LOAD
LOAD      M10517	// 02_-
AND       M10537	// STEP A¢Ò¡ÆC8
OR LOAD
LOAD      M10518	// 02_-
AND       M10538	// STEP A¢Ò¡ÆC9
OR LOAD
LOAD      M10519	// 02_-
AND       M10539	// STEP A¢Ò¡ÆC10
OR LOAD
LOAD      M1051A	// 02_-
AND       M1053A	// STEP A¢Ò¡ÆC11
OR LOAD
LOAD      M1051B	// 02_-
AND       M1053B	// STEP A¢Ò¡ÆC12
OR LOAD
LOAD      M1051C	// 02_-
AND       M1053C	// STEP A¢Ò¡ÆC13
OR LOAD
LOAD      M1051D	// 02_-
AND       M1053D	// STEP A¢Ò¡ÆC14
OR LOAD
LOAD      M1051E	// 02_-
AND       M1053E	// STEP A¢Ò¡ÆC15
OR LOAD
LOAD      M1051F	// 02_AU¥ì¢¯ STEP END
AND       M1053F	// STEP A¢Ò¡ÆC16
OR LOAD
AND LOAD
AND NOT   T1020	// L_2nd MAND STEP DELAY TM
AND       M10580	// L_2nd MAND CYCLE RUN
TON       T1020 D010150	// L_2nd MAND STEP DELAY TM
// ======================== SHIFT ==========================
; L47
LOAD      T1020	// L_2nd MAND STEP DELAY TM
DBSFLP    M1051 1
INCP      Z012

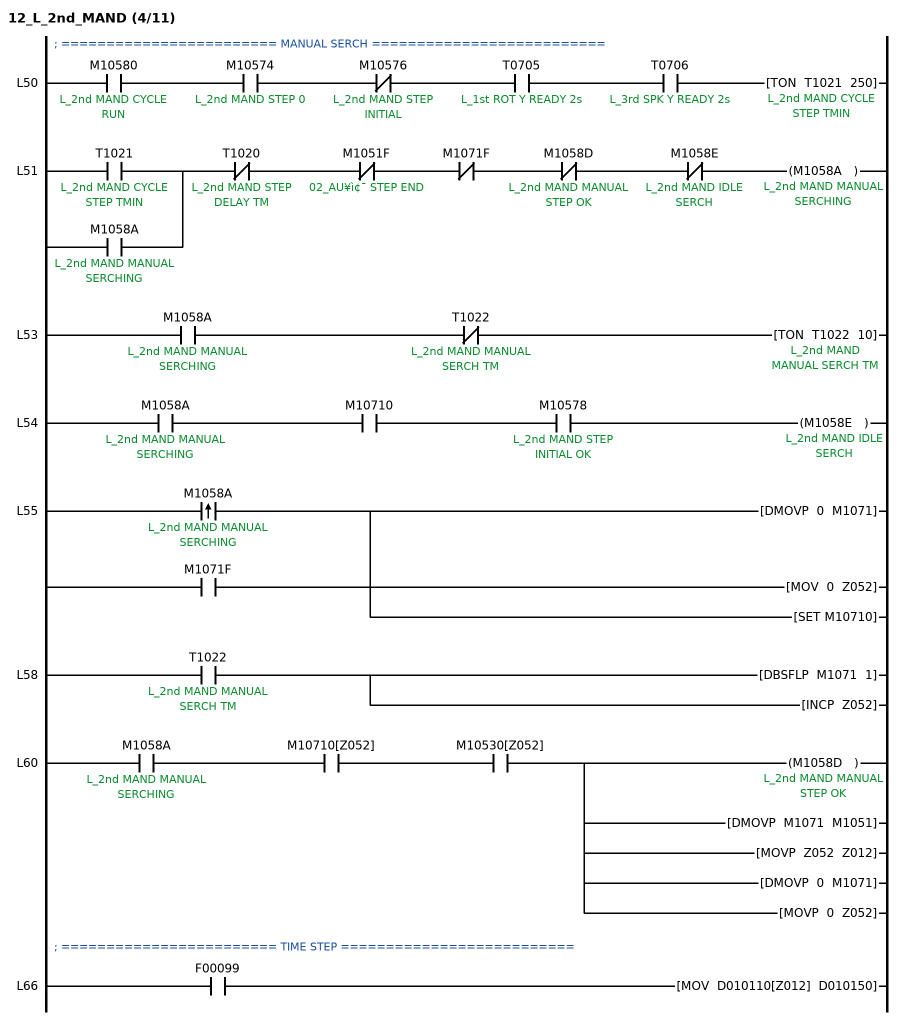
// ======================== MANUAL SERCH ==========================
; L50
LOAD      M10580	// L_2nd MAND CYCLE RUN
AND       M10574	// L_2nd MAND STEP 0
AND NOT   M10576	// L_2nd MAND STEP INITIAL
AND       T0705	// L_1st ROT Y READY 2s
AND       T0706	// L_3rd SPK Y READY 2s
TON       T1021 250	// L_2nd MAND CYCLE STEP TMIN
; L51
LOAD      T1021	// L_2nd MAND CYCLE STEP TMIN
OR        M1058A	// L_2nd MAND MANUAL SERCHING
AND NOT   T1020	// L_2nd MAND STEP DELAY TM
AND NOT   M1051F	// 02_AU¥ì¢¯ STEP END
AND NOT   M1071F
AND NOT   M1058D	// L_2nd MAND MANUAL STEP OK
AND NOT   M1058E	// L_2nd MAND IDLE SERCH
OUT       M1058A	// L_2nd MAND MANUAL SERCHING
; L53
LOAD      M1058A	// L_2nd MAND MANUAL SERCHING
AND NOT   T1022	// L_2nd MAND MANUAL SERCH TM
TON       T1022 10	// L_2nd MAND MANUAL SERCH TM
; L54
LOAD      M1058A	// L_2nd MAND MANUAL SERCHING
AND       M10710
AND       M10578	// L_2nd MAND STEP INITIAL OK
OUT       M1058E	// L_2nd MAND IDLE SERCH
; L55
LOADP     M1058A	// L_2nd MAND MANUAL SERCHING
OR        M1071F
DMOVP     0 M1071
MOV       0 Z052
SET       M10710
; L58
LOAD      T1022	// L_2nd MAND MANUAL SERCH TM
DBSFLP    M1071 1
INCP      Z052
; L60
LOAD      M1058A	// L_2nd MAND MANUAL SERCHING
AND       M10710[Z052]
AND       M10530[Z052]
OUT       M1058D	// L_2nd MAND MANUAL STEP OK
DMOVP     M1071 M1051
MOVP      Z052 Z012
DMOVP     0 M1071
MOVP      0 Z052
// ======================== TIME STEP ==========================
; L66
LOAD      F00099
MOV       D010110[Z012] D010150

